(* CODESYS project MC516.project
   CompiledLibraryCompatibilityVersion: LeadSysStudio V3.5 SP15 Patch 4
   Title: MC516

Project tree, tasks and I/O mapping:
  Device : MC516, Leadshine Technology Co., Ltd., order no. 516101, version 3.5.15.40
      settings: RetainMode = 0; RetainStartAddr = 20480; RetainEndAddr = 524288; RetainSize = 524288
    application Application
      libraries: Standard, * (System); VisuDialogs, * (System)
      task EtherCAT_Master_Leadshine_A (cyclic, interval 2000 µs, priority 0) calls EtherCAT_Master_Leadshine_A.EtherCAT_Task, M
      program M [ST]: io, motion, save_check, save_apply, work
      DataMain/
        data type HMIData
        data type SaveData
      function block AxisFB [ST]: calculate_home_delta_μ, follow
      Enum/
        data type State
        data type JogType
      Object/
        data type Button
        data type Cylinder
        data type AxisEC
        data type AxisECFollow
        data type AirBurst
        data type Problem
      function StateNext [ST]
      DataWork/
        data type SupplyData
        data type WorkData
        data type TapData
      function block TapFB [ST]
      visualisation Visualization
      function block SupplyFB [ST]
      Symbols
      function block SimpleMotion [ST]
      trace Trace (task EtherCAT_Master_Leadshine_A): M.tap_data.deviation
      function block AxisFBSetTorqueLimit [ST]
      global variables PersistentVars
    Resource Usage
    Device Diagnose
    Network Configuration
      LocalBus Config
    SoftMotion General Axis Pool
      AxisTap : Axis, 3S - Smart Software Solutions GmbH, order no. 1805, version 4.0.0.0
          settings: wDriveID = 3; eRampType = 3
    High_Speed_IO_Module : High Speed IO, Leadshine Technology Co., Ltd., version 3.5.15.40
        settings: HS_IO_Mode_0.High In IO Mode 0 = 196611; HS_IO_Mode_0.High In IO Mode 2 = 196611; Counter_Mask = 5; Ioin_Mask = 19; HS counter 1.Counter_CountMode = 1; HS counter 2.Counter_CountMode = 1; HS counter 3.Counter_SetWorkMode = 2; HS counter 3.Counter_CountMode = 1; InputFilter Para.Time_In0 = 2; InputFilter Para.Time_In1 = 2; InputFilter Para.Time_In4 = 2
        unmapped channels: Genral_IO_IN, Genral_IO_Out
    LocalBus_Master_Module : LocalBus Master, Leadshine Technology Co., Ltd., version 3.5.15.40
    EtherCAT_Master_Leadshine_A : EtherCAT Master SoftMotion, 3S - Smart Software Solutions GmbH, version 3.5.16.30
        settings: MasterCycleTime = 2000; NetworkName = 'ecat'; SelectNetworkByName = TRUE; SrcAddress1 = 10; SrcAddress2 = 889192738
      XINJE_DS5C1_CoE_Drive_Rev4_0_2 : XINJE-DS5C1 EtherCAT(CoE) Drive Rev4.0 v3.7.70, Xinje Electronics, Inc., order no. XINJE-DS5C1 CoE Drive Rev4.0, version Revision=16#20201207
          settings: Number of Inputs = 6; Number of Infos about Inputs = 6; StationAlias = 4; Sync.Length = 17; FMMU.Length = 17; DC sync0 cycletime = 2000; DC sync1 cycletime = 2000; Number of SDO = 4; Interpolation time period.Value = 2; Homing method.Index = 16#0000; Homing method.Subindex = 16#00; Homing method.Size = 0; Homing method.AbortIfError = FALSE; Homing method.JumpToLine = FALSE; Homing method.Line = 0; Homing method.CompleteAccess = False; RxTxPdo.NumberofEntries = 6; RxTxPdo.Index = 16#1A00; RxTxPdo.DependOnSlot = False; RxTxPdo.DependOnSlotGroup = False; RxTxPdo.OverwrittenByModule = False; Status Word.Offset = 0; Status Word.DependOnSlot = False; Status Word.DependOnSlotGroup = False; ActualPosition.Offset = 0; ActualPosition.DependOnSlot = False; ActualPosition.DependOnSlotGroup = False; Velocity actual value.Offset = 0; Velocity actual value.DependOnSlot = False; Velocity actual value.DependOnSlotGroup = False; ActualTorque.Offset = 0; ActualTorque.DependOnSlot = False; ActualTorque.DependOnSlotGroup = False; ModeOfOperationDisplay.Offset = 0; ModeOfOperationDisplay.DependOnSlot = False; ModeOfOperationDisplay.DependOnSlotGroup = False; Index = 16#5000; SubIndex = 0; Size = 32; Offset = 0;
            DependOnSlot = False; DependOnSlotGroup = False; Status Word.Default = ''; Status Word.Comment = ''; ActualPosition.Default = ''; ActualPosition.Comment = ''; Velocity actual value.Default = ''; Velocity actual value.Comment = ''; ActualTorque.Default = ''; ActualTorque.Comment = ''; ModeOfOperationDisplay.Default = ''; ModeOfOperationDisplay.Comment = ''; Name = 'Encode Single Position'; DataType = 'DINT'; Default = ''; Comment = ''
          unmapped channels: Control Word, TargetPosition, TargetVelocity, TargetTorque, ModeOfOperation, Status Word, ActualPosition, Velocity actual value, ActualTorque, ModeOfOperationDisplay, Encode Single Position
        Axis_2 : Axis, 3S - Smart Software Solutions GmbH, order no. 0, version 4.6.1.0
            settings: wDriveID = 7; dwRatioTechUnitsDenom = 1; eRampType = 3; Number of pulses for one revolution = 131072; The displacement for one revolution of the workbench = 131072; Gear ratio molecule = 1; Gear ratio denominator = 1; ScalingIncs = 131072; AdrOffset_8010 = 36; BitOffset_8010 = 0; BitLength_8010 = 16; Address_8010 = '%QW18'; Type_8010 = 'UINT'; AddressPointer_8010 = ADR(%QW18); AdrOffset_8020 = 40; BitOffset_8020 = 0; BitLength_8020 = 32; Address_8020 = '%QD10'; Type_8020 = 'DINT'; AddressPointer_8020 = ADR(%QD10); AdrOffset_8030 = 44; BitOffset_8030 = 0; BitLength_8030 = 32; Address_8030 = '%QD11'; Type_8030 = 'DINT'; AddressPointer_8030 = ADR(%QD11); AdrOffset_8040 = 48; BitOffset_8040 = 0; BitLength_8040 = 16; Address_8040 = '%QW24'; Type_8040 = 'INT'; AddressPointer_8040 = ADR(%QW24); AdrOffset_8050 = 50; BitOffset_8050 = 0; BitLength_8050 = 8; Address_8050 = '%QB50'; Type_8050 = 'SINT'; AddressPointer_8050 = ADR(%QB50); AdrOffset_8060 = 4294967295; BitOffset_8060 = 0;
              BitLength_8060 = 0; Address_8060 = ''; Type_8060 = ''; AddressPointer_8060 = 0; AdrOffset_8070 = 4294967295; BitOffset_8070 = 0; BitLength_8070 = 0; Address_8070 = ''; Type_8070 = ''; AddressPointer_8070 = 0; AdrOffset_8080 = 4294967295; BitOffset_8080 = 0; BitLength_8080 = 0; Address_8080 = ''; Type_8080 = ''; AddressPointer_8080 = 0; AdrOffset_8090 = 4294967295; BitOffset_8090 = 0; BitLength_8090 = 0; Address_8090 = ''; Type_8090 = ''; AddressPointer_8090 = 0; AdrOffset_8510 = 44; BitOffset_8510 = 0; BitLength_8510 = 16; Address_8510 = '%IW22'; Type_8510 = 'UINT'; AddressPointer_8510 = ADR(%IW22); AdrOffset_8520 = 48; BitOffset_8520 = 0; BitLength_8520 = 32; Address_8520 = '%ID12'; Type_8520 = 'DINT'; AddressPointer_8520 = ADR(%ID12); AdrOffset_8530 = 52; BitOffset_8530 = 0; BitLength_8530 = 32; Address_8530 = '%ID13'; Type_8530 = 'DINT'; AddressPointer_8530 = ADR(%ID13);
              AdrOffset_8540 = 56; BitOffset_8540 = 0; BitLength_8540 = 16; Address_8540 = '%IW28'; Type_8540 = 'INT'; AddressPointer_8540 = ADR(%IW28); AdrOffset_8550 = 58; BitOffset_8550 = 0; BitLength_8550 = 8; Address_8550 = '%IB58'; Type_8550 = 'SINT'; AddressPointer_8550 = ADR(%IB58); AdrOffset_8560 = 4294967295; BitOffset_8560 = 0; BitLength_8560 = 0; Address_8560 = ''; Type_8560 = ''; AddressPointer_8560 = 0; AdrOffset_8570 = 4294967295; BitOffset_8570 = 0; BitLength_8570 = 0; Address_8570 = ''; Type_8570 = ''; AddressPointer_8570 = 0; AdrOffset_8580 = 4294967295; BitOffset_8580 = 0; BitLength_8580 = 0; Address_8580 = ''; Type_8580 = ''; AddressPointer_8580 = 0; AdrOffset_8590 = 4294967295; BitOffset_8590 = 0; BitLength_8590 = 0; Address_8590 = ''; Type_8590 = ''; AddressPointer_8590 = 0; AdrOffset_8600 = 4294967295; BitOffset_8600 = 0; BitLength_8600 = 0; Address_8600 = '';
              Type_8600 = ''; AddressPointer_8600 = 0; AdrOffset_8600 = 4294967295; BitOffset_8600 = 0; BitLength_8600 = 0; Address_8610 = ''; Type_8610 = ''; AddressPointer_8610 = 0; AdrOffset_8620 = 4294967295; BitOffset_8620 = 0; BitLength_8620 = 0; Address_8620 = ''; Type_8620 = ''; AddressPointer_8620 = 0
      XINJE_DS5C1_CoE_Drive_Rev4_0_1 : XINJE-DS5C1 EtherCAT(CoE) Drive Rev4.0 v3.7.70, Xinje Electronics, Inc., order no. XINJE-DS5C1 CoE Drive Rev4.0, version Revision=16#20201207
          settings: Number of Inputs = 6; Number of Infos about Inputs = 6; StationAlias = 3; Sync.Length = 17; FMMU.Length = 17; DC sync0 cycletime = 2000; DC sync1 cycletime = 2000; Number of SDO = 4; Interpolation time period.Value = 2; Homing method.Index = 16#0000; Homing method.Subindex = 16#00; Homing method.Size = 0; Homing method.AbortIfError = FALSE; Homing method.JumpToLine = FALSE; Homing method.Line = 0; Homing method.CompleteAccess = False; RxTxPdo.NumberofEntries = 6; RxTxPdo.Index = 16#1A00; RxTxPdo.DependOnSlot = False; RxTxPdo.DependOnSlotGroup = False; RxTxPdo.OverwrittenByModule = False; Status Word.Offset = 0; Status Word.DependOnSlot = False; Status Word.DependOnSlotGroup = False; ActualPosition.Offset = 0; ActualPosition.DependOnSlot = False; ActualPosition.DependOnSlotGroup = False; Velocity actual value.Offset = 0; Velocity actual value.DependOnSlot = False; Velocity actual value.DependOnSlotGroup = False; ActualTorque.Offset = 0; ActualTorque.DependOnSlot = False; ActualTorque.DependOnSlotGroup = False; ModeOfOperationDisplay.Offset = 0; ModeOfOperationDisplay.DependOnSlot = False; ModeOfOperationDisplay.DependOnSlotGroup = False; Index = 16#5000; SubIndex = 0; Size = 32; Offset = 0;
            DependOnSlot = False; DependOnSlotGroup = False; Status Word.Default = ''; Status Word.Comment = ''; ActualPosition.Default = ''; ActualPosition.Comment = ''; Velocity actual value.Default = ''; Velocity actual value.Comment = ''; ActualTorque.Default = ''; ActualTorque.Comment = ''; ModeOfOperationDisplay.Default = ''; ModeOfOperationDisplay.Comment = ''; Name = 'Encode Single Position'; DataType = 'DINT'; Default = ''; Comment = ''
          unmapped channels: Control Word, TargetPosition, TargetVelocity, TargetTorque, ModeOfOperation, Status Word, ActualPosition, Velocity actual value, ActualTorque, ModeOfOperationDisplay, Encode Single Position
        Axis_1 : Axis, 3S - Smart Software Solutions GmbH, order no. 0, version 4.6.1.0
            settings: wDriveID = 6; dwRatioTechUnitsDenom = 1; eRampType = 3; Number of pulses for one revolution = 131072; The displacement for one revolution of the workbench = 131072; Gear ratio molecule = 1; Gear ratio denominator = 1; ScalingIncs = 131072; AdrOffset_8010 = 20; BitOffset_8010 = 0; BitLength_8010 = 16; Address_8010 = '%QW10'; Type_8010 = 'UINT'; AddressPointer_8010 = ADR(%QW10); AdrOffset_8020 = 24; BitOffset_8020 = 0; BitLength_8020 = 32; Address_8020 = '%QD6'; Type_8020 = 'DINT'; AddressPointer_8020 = ADR(%QD6); AdrOffset_8030 = 28; BitOffset_8030 = 0; BitLength_8030 = 32; Address_8030 = '%QD7'; Type_8030 = 'DINT'; AddressPointer_8030 = ADR(%QD7); AdrOffset_8040 = 32; BitOffset_8040 = 0; BitLength_8040 = 16; Address_8040 = '%QW16'; Type_8040 = 'INT'; AddressPointer_8040 = ADR(%QW16); AdrOffset_8050 = 34; BitOffset_8050 = 0; BitLength_8050 = 8; Address_8050 = '%QB34'; Type_8050 = 'SINT'; AddressPointer_8050 = ADR(%QB34); AdrOffset_8060 = 4294967295; BitOffset_8060 = 0;
              BitLength_8060 = 0; Address_8060 = ''; Type_8060 = ''; AddressPointer_8060 = 0; AdrOffset_8070 = 4294967295; BitOffset_8070 = 0; BitLength_8070 = 0; Address_8070 = ''; Type_8070 = ''; AddressPointer_8070 = 0; AdrOffset_8080 = 4294967295; BitOffset_8080 = 0; BitLength_8080 = 0; Address_8080 = ''; Type_8080 = ''; AddressPointer_8080 = 0; AdrOffset_8090 = 4294967295; BitOffset_8090 = 0; BitLength_8090 = 0; Address_8090 = ''; Type_8090 = ''; AddressPointer_8090 = 0; AdrOffset_8510 = 24; BitOffset_8510 = 0; BitLength_8510 = 16; Address_8510 = '%IW12'; Type_8510 = 'UINT'; AddressPointer_8510 = ADR(%IW12); AdrOffset_8520 = 28; BitOffset_8520 = 0; BitLength_8520 = 32; Address_8520 = '%ID7'; Type_8520 = 'DINT'; AddressPointer_8520 = ADR(%ID7); AdrOffset_8530 = 32; BitOffset_8530 = 0; BitLength_8530 = 32; Address_8530 = '%ID8'; Type_8530 = 'DINT'; AddressPointer_8530 = ADR(%ID8);
              AdrOffset_8540 = 36; BitOffset_8540 = 0; BitLength_8540 = 16; Address_8540 = '%IW18'; Type_8540 = 'INT'; AddressPointer_8540 = ADR(%IW18); AdrOffset_8550 = 38; BitOffset_8550 = 0; BitLength_8550 = 8; Address_8550 = '%IB38'; Type_8550 = 'SINT'; AddressPointer_8550 = ADR(%IB38); AdrOffset_8560 = 4294967295; BitOffset_8560 = 0; BitLength_8560 = 0; Address_8560 = ''; Type_8560 = ''; AddressPointer_8560 = 0; AdrOffset_8570 = 4294967295; BitOffset_8570 = 0; BitLength_8570 = 0; Address_8570 = ''; Type_8570 = ''; AddressPointer_8570 = 0; AdrOffset_8580 = 4294967295; BitOffset_8580 = 0; BitLength_8580 = 0; Address_8580 = ''; Type_8580 = ''; AddressPointer_8580 = 0; AdrOffset_8590 = 4294967295; BitOffset_8590 = 0; BitLength_8590 = 0; Address_8590 = ''; Type_8590 = ''; AddressPointer_8590 = 0; AdrOffset_8600 = 4294967295; BitOffset_8600 = 0; BitLength_8600 = 0; Address_8600 = '';
              Type_8600 = ''; AddressPointer_8600 = 0; AdrOffset_8600 = 4294967295; BitOffset_8600 = 0; BitLength_8600 = 0; Address_8610 = ''; Type_8610 = ''; AddressPointer_8610 = 0; AdrOffset_8620 = 4294967295; BitOffset_8620 = 0; BitLength_8620 = 0; Address_8620 = ''; Type_8620 = ''; AddressPointer_8620 = 0
      XINJE_DS5C1_CoE_Drive_Rev4_0 : XINJE-DS5C1 EtherCAT(CoE) Drive Rev4.0 v3.7.70, Xinje Electronics, Inc., order no. XINJE-DS5C1 CoE Drive Rev4.0, version Revision=16#20201207
          settings: Number of Inputs = 6; Number of Infos about Inputs = 6; StationAlias = 1; Sync.Length = 17; FMMU.Length = 17; DC sync0 cycletime = 2000; DC sync1 cycletime = 2000; Number of SDO = 4; Interpolation time period.Value = 2; Homing method.Index = 16#0000; Homing method.Subindex = 16#00; Homing method.Size = 0; Homing method.AbortIfError = FALSE; Homing method.JumpToLine = FALSE; Homing method.Line = 0; Homing method.CompleteAccess = False; RxTxPdo.NumberofEntries = 6; RxTxPdo.Index = 16#1A00; RxTxPdo.DependOnSlot = False; RxTxPdo.DependOnSlotGroup = False; RxTxPdo.OverwrittenByModule = False; Status Word.Offset = 0; Status Word.DependOnSlot = False; Status Word.DependOnSlotGroup = False; ActualPosition.Offset = 0; ActualPosition.DependOnSlot = False; ActualPosition.DependOnSlotGroup = False; Velocity actual value.Offset = 0; Velocity actual value.DependOnSlot = False; Velocity actual value.DependOnSlotGroup = False; ActualTorque.Offset = 0; ActualTorque.DependOnSlot = False; ActualTorque.DependOnSlotGroup = False; ModeOfOperationDisplay.Offset = 0; ModeOfOperationDisplay.DependOnSlot = False; ModeOfOperationDisplay.DependOnSlotGroup = False; Index = 16#5000; SubIndex = 0; Size = 32; Offset = 0;
            DependOnSlot = False; DependOnSlotGroup = False; Status Word.Default = ''; Status Word.Comment = ''; ActualPosition.Default = ''; ActualPosition.Comment = ''; Velocity actual value.Default = ''; Velocity actual value.Comment = ''; ActualTorque.Default = ''; ActualTorque.Comment = ''; ModeOfOperationDisplay.Default = ''; ModeOfOperationDisplay.Comment = ''; Name = 'Encode Single Position'; DataType = 'DINT'; Default = ''; Comment = ''
          unmapped channels: Control Word, TargetPosition, TargetVelocity, TargetTorque, ModeOfOperation, Status Word, ActualPosition, Velocity actual value, ActualTorque, ModeOfOperationDisplay, Encode Single Position
        Axis : Axis, 3S - Smart Software Solutions GmbH, order no. 0, version 4.6.1.0
            settings: wDriveID = 4; dwRatioTechUnitsDenom = 1; eRampType = 3; Number of pulses for one revolution = 131072; The displacement for one revolution of the workbench = 131072; Gear ratio molecule = 1; Gear ratio denominator = 1; ScalingIncs = 131072; AdrOffset_8010 = 4; BitOffset_8010 = 0; BitLength_8010 = 16; Address_8010 = '%QW2'; Type_8010 = 'UINT'; AddressPointer_8010 = ADR(%QW2); AdrOffset_8020 = 8; BitOffset_8020 = 0; BitLength_8020 = 32; Address_8020 = '%QD2'; Type_8020 = 'DINT'; AddressPointer_8020 = ADR(%QD2); AdrOffset_8030 = 12; BitOffset_8030 = 0; BitLength_8030 = 32; Address_8030 = '%QD3'; Type_8030 = 'DINT'; AddressPointer_8030 = ADR(%QD3); AdrOffset_8040 = 16; BitOffset_8040 = 0; BitLength_8040 = 16; Address_8040 = '%QW8'; Type_8040 = 'INT'; AddressPointer_8040 = ADR(%QW8); AdrOffset_8050 = 18; BitOffset_8050 = 0; BitLength_8050 = 8; Address_8050 = '%QB18'; Type_8050 = 'SINT'; AddressPointer_8050 = ADR(%QB18); AdrOffset_8060 = 4294967295; BitOffset_8060 = 0;
              BitLength_8060 = 0; Address_8060 = ''; Type_8060 = ''; AddressPointer_8060 = 0; AdrOffset_8070 = 4294967295; BitOffset_8070 = 0; BitLength_8070 = 0; Address_8070 = ''; Type_8070 = ''; AddressPointer_8070 = 0; AdrOffset_8080 = 4294967295; BitOffset_8080 = 0; BitLength_8080 = 0; Address_8080 = ''; Type_8080 = ''; AddressPointer_8080 = 0; AdrOffset_8090 = 4294967295; BitOffset_8090 = 0; BitLength_8090 = 0; Address_8090 = ''; Type_8090 = ''; AddressPointer_8090 = 0; AdrOffset_8510 = 4; BitOffset_8510 = 0; BitLength_8510 = 16; Address_8510 = '%IW2'; Type_8510 = 'UINT'; AddressPointer_8510 = ADR(%IW2); AdrOffset_8520 = 8; BitOffset_8520 = 0; BitLength_8520 = 32; Address_8520 = '%ID2'; Type_8520 = 'DINT'; AddressPointer_8520 = ADR(%ID2); AdrOffset_8530 = 12; BitOffset_8530 = 0; BitLength_8530 = 32; Address_8530 = '%ID3'; Type_8530 = 'DINT'; AddressPointer_8530 = ADR(%ID3);
              AdrOffset_8540 = 16; BitOffset_8540 = 0; BitLength_8540 = 16; Address_8540 = '%IW8'; Type_8540 = 'INT'; AddressPointer_8540 = ADR(%IW8); AdrOffset_8550 = 18; BitOffset_8550 = 0; BitLength_8550 = 8; Address_8550 = '%IB18'; Type_8550 = 'SINT'; AddressPointer_8550 = ADR(%IB18); AdrOffset_8560 = 4294967295; BitOffset_8560 = 0; BitLength_8560 = 0; Address_8560 = ''; Type_8560 = ''; AddressPointer_8560 = 0; AdrOffset_8570 = 4294967295; BitOffset_8570 = 0; BitLength_8570 = 0; Address_8570 = ''; Type_8570 = ''; AddressPointer_8570 = 0; AdrOffset_8580 = 4294967295; BitOffset_8580 = 0; BitLength_8580 = 0; Address_8580 = ''; Type_8580 = ''; AddressPointer_8580 = 0; AdrOffset_8590 = 4294967295; BitOffset_8590 = 0; BitLength_8590 = 0; Address_8590 = ''; Type_8590 = ''; AddressPointer_8590 = 0; AdrOffset_8600 = 4294967295; BitOffset_8600 = 0; BitLength_8600 = 0; Address_8600 = '';
              Type_8600 = ''; AddressPointer_8600 = 0; AdrOffset_8600 = 4294967295; BitOffset_8600 = 0; BitLength_8600 = 0; Address_8610 = ''; Type_8610 = ''; AddressPointer_8610 = 0; AdrOffset_8620 = 4294967295; BitOffset_8620 = 0; BitLength_8620 = 0; Address_8620 = ''; Type_8620 = ''; AddressPointer_8620 = 0
  text list GlobalTextList
*)

// Device/Application/DataMain/HMIData
{ attribute 'pack_mode' := ''}
TYPE HMIData :
STRUCT
	//
	sv: SaveData;
	sv_trigger: BOOL;
	sv_need_check: BOOL;
	sv_need: BOOL;
	//
	plc_ready: BOOL;
	hmi_ready: BOOL;
	run: BOOL;
	stop: BOOL;
	home: BOOL;
	problem_fix: ARRAY[0..7] OF BOOL;
	//
	supply_test: BOOL;
	supply_clamp: BOOL;
	supply_extract_down: BOOL;
	supply_extract_pull: BOOL;
	tap_lubricate: BOOL;
	supply_clean: BOOL;
	jog_micro_per_sec_or_rev: UINT;
	jog_n: BOOL;
	jog_p: BOOL;
	//
	view_input: ARRAY[0..15] OF BOOL;
	view_output: ARRAY[0..15] OF BOOL;
	//
	view_can_run: BOOL;
	view_can_stop: BOOL;
	view_can_home: BOOL;
	view_auto: BOOL;
	view_manual: BOOL;
	//
	view_axis_encoder: ARRAY[0..2] OF DINT;
	view_axis_micro: ARRAY[0..2] OF DINT;
	view_axis_mNm: ARRAY[0..2] OF UDINT;
	//
	view_load: UINT;
	view_problem: ARRAY[0..7] OF BOOL;
	view_tap_deviation_micron: UINT;
	view_cycle_count: UDINT;
	view_cycle_time_msec: UDINT;
	//
	view_state: ARRAY[0..4] OF INT;
END_STRUCT
END_TYPE

// Device/Application/DataMain/SaveData
{ attribute 'pack_mode' := ''}
TYPE SaveData :
STRUCT
	set_done: BOOL;
	////////
	//SAME//
	////////
	cylinder_n_delay_msec: ARRAY[0..2] OF UINT;
	cylinder_p_delay_msec: ARRAY[0..2] OF UINT;
	air_burst_delay_msec: ARRAY[0..1] OF UINT;
	//
	// (a) increments        <> (d) motor turns
	// (b) motor turns       <> (e) gear output turns
	// (c) gear output turns <> (f) units in application
	// .iRatioTechUnitsNum = gear_num = gear_dir * d * e * f 
	// .dwRatioTechUnitsDenom = gear_den = a * b * c
	max_rpm: ARRAY[0..2] OF UINT;
	gear_num: ARRAY[0..2] OF DINT;
	gear_den: ARRAY[0..2] OF DINT;
	gear_dir: ARRAY[0..2] OF BOOL;
	home_torque_mNm: ARRAY[0..2] OF UINT;
	home_encoder_value_recorded: BOOL;
	home_encoder_value: ARRAY[0..2] OF DINT;
	max_micro_recorded: BOOL;
	max_micro: ARRAY[0..2] OF DINT;
	overload_hold_torque_factor: ARRAY[0..2] OF UINT;
	overload_hold_torque_time_msec: ARRAY[0..2] OF UINT;
	overload_instant_torque_factor: ARRAY[0..2] OF UINT;
	ramp_time_msec: ARRAY[0..2] OF UINT;
	jerk_factor: ARRAY[0..2] OF UINT;
	///////////
	//MACHINE//
	///////////
	supply_micro_per_sec: UDINT;
	//
	tap_begin_micron: UDINT; // vị trí bắt đầu taro
	tap_depth_micron: UDINT; // độ sâu từ vị trí bắt đầu taro
	tap_micron_per_rev: UDINT; // bước ren μm
	tap_rpm: UDINT; // tốc độ taro
	tap_backlash_micro: UINT; // độ rơ micro vòng
	tap_deviation_micron_max: UINT;
END_STRUCT
END_TYPE

// Device/Application/Enum/State
{attribute 'qualified_only'}
{attribute 'strict'}
TYPE State :
(
	NONE := 0,
	RST := 1,
	RST_DONE := 50,
	HOME := 51,
	HOME_FORWARD := 71,
	HOME_DONE := 90,
	HOME_OFFSET := 91,
	HOME_OFFSET_DONE := 99,
	READY := 100,
	RUN := 101,
	RUN_ING := 200
);
END_TYPE

// Device/Application/Object/Button
{ attribute 'pack_mode' := ''}
TYPE Button :
STRUCT
	on: BOOL;
	rise: R_TRIG;
	rise_physical: R_TRIG;
	fall: F_TRIG;
	fall_physical: F_TRIG;
	timer: TON;
END_STRUCT
END_TYPE

// Device/Application/Object/Cylinder
{ attribute 'pack_mode' := ''}
TYPE Cylinder :
STRUCT
	on: BOOL;
	n_timer: TON;
	p_timer: TON;
END_STRUCT
END_TYPE

// Device/Application/Object/AxisEC
{ attribute 'pack_mode' := ''}
TYPE AxisEC :
STRUCT
	///////
	//REF//
	///////
	ref: POINTER TO SM3_Drive_ETC_DS402_CyclicSync.AXIS_REF_ETC_DS402_CS;
	read: POINTER TO SMC3_ETC_ReadParameter_CoE;
	write: POINTER TO SMC3_ETC_WriteParameter_CoE;
	read_status: POINTER TO MC_ReadStatus;
	set_mode: POINTER TO SMC_SetControllerMode;
	power: POINTER TO MC_Power;
	reset: POINTER TO MC_Reset;
	stop: POINTER TO MC_Stop;
	inch: POINTER TO SMC_Inch;
	fsv: POINTER TO SMC_FollowSetValues;
	sp: POINTER TO MC_SetPosition;
	mabs: POINTER TO MC_MoveAbsolute;
	set_torque_limit: AxisFBSetTorqueLimit;
	////////
	//DATA//
	////////
	encoder_resolution: DINT;
	torque_rated_Nm: LREAL;
	encoder_single_position: DINT;
	///////////
	//PROCESS//
	///////////
	state: INT;
	torque_Nm: LREAL;
	torque_Nm_abs: LREAL;
	overload: BOOL;
	overload_check: BOOL;
	overload_hold_torque_Nm: LREAL;
	overload_hold_torque_timer: TON;
	overload_instant_torque_Nm: LREAL;
	//home
	home_done: BOOL; // = TRUE khi về gốc thành công, chỉ về gốc khi bật máy
	home_done_forward_ignore: BOOL;
	home_to_encoder: BOOL; //
	home_torque_Nm: LREAL;
	home_hit_timer: TON;
	home_hit_test: BOOL;
	home_offset_absolute_μ: LREAL; // vị trí từ điểm va chạm đến gốc tuyệt đối, xem hàm save_apply()
	home_back_μ_per_sec: LREAL; // tốc độ lùi về lấy gốc
	home_forward_μ_per_sec: LREAL; // tốc độ tiến sau khi lấy gốc xong
	home_offset_μ: LREAL; // giá trị này để thực hiện lệnh state = State.HOME_OFFSET ở trong AxisLinearFB
	home_encoder_value_recorded: BOOL;
	home_encoder_value_save: POINTER TO DINT; // pointer tới giá trị ở save data
	home_encoder_delta: DINT;
	home_delta_μ: LREAL;
	//
	ramp_time_sec: LREAL;
	jerk_factor: LREAL;
	//
	jog_type: JogType;
	jog_delta: LREAL;
	jog_velocity: LREAL;
	jog_acceleration: LREAL;
	max_μ_recorded: BOOL;
	max_μ_save: POINTER TO DINT;
	max_μ: LREAL; // giới hạn vị trí tối đa có thể di chuyển từ gốc tuyệt đối
	max_μ_per_sec: LREAL; // giới hạn tốc độ tối đa
	//run
	target_position_μ: LREAL; // sử dụng cho state = State.RUN ở trong AxisLinearFB
	target_velocity_μ_per_sec: LREAL; // sử dụng cho state = State.RUN ở trong AxisLinearFB
END_STRUCT
END_TYPE

// Device/Application/DataWork/SupplyData
{ attribute 'pack_mode' := ''}
TYPE SupplyData :
STRUCT
	state: INT;
	state_extract: INT;
	axis: AxisEC;
	axis_fb: AxisFB;
	//
	input_air: BOOL;
	input_foil: BOOL;
	//
	no_air: Problem;
	foil_stuck: Problem;
	clamp: Cylinder;
	extract_down: Cylinder;
	extract_pull: Cylinder;
	clean: AirBurst;
	//
	index_count: LREAL;
	μ_per_sec: LREAL;
END_STRUCT
END_TYPE

// Device/Application/DataWork/WorkData
{ attribute 'pack_mode' := ''}
TYPE WorkData :
STRUCT
	state: INT;
	//
	input_run: Button;
	input_stop: Button;
	input_home: Button;
	//
	can_run: BOOL;
	can_stop: BOOL;
	can_home: BOOL;
	auto: Button;
	overload: Problem;
	alarm: BOOL;
	//
	supply_test: Button;
	//
	manual: BOOL;
	cycle_start_msec: ULINT;
	cycle_time_msec: UDINT;
END_STRUCT
END_TYPE

// Device/Application/DataWork/TapData
{ attribute 'pack_mode' := ''}
TYPE TapData :
STRUCT
	state: INT;
	axis_move: AxisEC;
	axis_move_fb: AxisFB;
	axis_move_follow_data: AxisECFollow;
	axis_spin: AxisEC;
	axis_spin_fb: AxisFB;
	axis_spin_follow_data: AxisECFollow;
	//
	axis_v: POINTER TO SM3_Basic.AXIS_REF_VIRTUAL_SM3;
	axis_v_power: MC_Power;
	axis_v_stop: MC_Stop;
	axis_v_inch: SMC_Inch;
	axis_v_sp: MC_SetPosition;
	axis_v_mabs: MC_MoveAbsolute;
	//
	begin_μm: LREAL;
	depth_μm: LREAL;
	μm_per_rev: LREAL;
	rps: LREAL;
	backlash_μ: LREAL;
	//
	lubricate: AirBurst;
	//
	deviation_μm: LREAL;
	deviation_μm_max: LREAL;
	deviation_overload: BOOL;
	//
	load: LREAL;
	load_sum: LREAL;
	load_count: LREAL;
	time_delta_sec: LREAL;
END_STRUCT
END_TYPE

// Device/Application/Object/AxisECFollow
TYPE AxisECFollow :
STRUCT
	target: POINTER TO SM3_Basic.AXIS_REF_SM3;
	ratio: LREAL;
	offset: LREAL;
	offset_motion: SimpleMotion;
	//
	self_begin: LREAL;
	target_begin: LREAL;
	target_delta: LREAL;
	//
	deviation: LREAL;
END_STRUCT
END_TYPE

// Device/Application/Object/AirBurst
TYPE AirBurst :
STRUCT
	on: BOOL;
	timer: TON;
END_STRUCT
END_TYPE

// Device/Application/Enum/JogType
{attribute 'qualified_only'}
{attribute 'strict'}
TYPE JogType :
(
	NONE := 0,
	INCH := 1, // inch function
	FSV := 2 // follow set value function
);
END_TYPE

// Device/Application/Object/Problem
TYPE Problem :
STRUCT
	on: BOOL;
	timer: TON;
	rise: R_TRIG;
	fix_rise: R_TRIG;
END_STRUCT
END_TYPE

// Device/Application/PersistentVars
{attribute 'qualified_only'}
VAR_GLOBAL PERSISTENT RETAIN
END_VAR
VAR_GLOBAL PERSISTENT
	M.save: SaveData;
END_VAR

// Device/Application/M
PROGRAM M
VAR
	time_msec_last: ULINT;
	time_msec : ULINT;
	time_delta_sec: LREAL;
	//
	axiss: ARRAY [0..2] OF POINTER TO SM3_Drive_ETC_DS402_CyclicSync.AXIS_REF_ETC_DS402_CS;
	// dùng pointer để dễ dàng thao tác với nhiều trục hơn, xem hàm motion()
	axiss_read: ARRAY[0..2] OF SMC3_ETC_ReadParameter_CoE;
	axiss_write: ARRAY[0..2] OF SMC3_ETC_WriteParameter_CoE;
	axiss_read_status: ARRAY[0..2] OF MC_ReadStatus;
	axiss_change_gearing_ratio: ARRAY[0..2] OF SMC_ChangeGearingRatio;
	axiss_reinit_drive: ARRAY[0..2] OF SMC3_ReinitDrive;
	axiss_set_mode: ARRAY[0..2] OF SMC_SetControllerMode;
	axiss_power: ARRAY[0..2] OF MC_Power; // bật tắt động cơ
	axiss_reset: ARRAY[0..2] OF MC_Reset; // reset lỗi
	axiss_stop: ARRAY[0..2] OF MC_Stop; // dừng
	axiss_inch: ARRAY[0..2] OF SMC_Inch;
	axiss_fsv: ARRAY[0..2] OF SMC_FollowSetValues;
	axiss_sp: ARRAY[0..2] OF MC_SetPosition;
	axiss_mabs: ARRAY[0..2] OF MC_MoveAbsolute;
	axiss_encoder_resolution: ARRAY[0..2] OF DINT;
	axiss_rated_torque_Nm: ARRAY[0..2] OF LREAL;
	axiss_max_rpm: ARRAY[0..2] OF UINT;
	axiss_max_μ_per_sec: ARRAY[0..2] OF LREAL;
	axiss_ready_all: BOOL;
	//
	state_main: INT;
	motion_active: BOOL;
	main_save: Button;
	supply_data: SupplyData;
	supply_fb: SupplyFB;
	tap_data: TapData;
	tap_fb: TapFB;
	work_data: WorkData;
	hmi: HMIData;
	//
	i: INT;
	j: INT;
	k: INT;
	axis_ec_i: POINTER TO AxisEC;
	axis_fb_i: POINTER TO AxisFB;
	cylinder_i: POINTER TO Cylinder;
	air_burst_i: POINTER TO AirBurst;
	//
	test: BOOL;
END_VAR

VAR CONSTANT
	c_axis_i_max: INT := 3 - 1;
	c_cylinder_i_max: INT := 3 - 1;
	c_air_burst_i_max: INT := 2 - 1;
END_VAR

VAR RETAIN
	cycle_count: UDINT;
	cycle_count_reset_time_msec: ULINT;
END_VAR

VAR PERSISTENT
	save: SaveData;
END_VAR

MC_SysLib.SysTimeRtc.SysTimeRtcHighResGet(pTimestamp:= time_msec);
time_delta_sec := ULINT_TO_LREAL(time_msec - time_msec_last) * 1E-3;
time_msec_last := time_msec;
hmi.view_state[0] := state_main;
IF motion_active THEN
	motion();
END_IF
CASE state_main OF
	State.NONE: // khi khởi động thì state_main = 0 tức là = State.NONE
		axiss[0] := ADR(Axis); // k = ADR(x) viết tắt cho "address of x" là hàm để lấy giá trị con trỏ (pointer) về biến x
		axiss[1] := ADR(Axis_1); // ví dụ muốn thay đổi giá trị của x ta sẽ viết k^ = 12345
		axiss[2] := ADR(Axis_2);
		axiss_change_gearing_ratio[0].iMovementType := SMC_MOVEMENTTYPE.rotary;
		axiss_change_gearing_ratio[1].iMovementType := SMC_MOVEMENTTYPE.linear;
		axiss_change_gearing_ratio[2].iMovementType := SMC_MOVEMENTTYPE.linear;
		axiss_change_gearing_ratio[0].fPositionPeriod := 1_000;
		axiss_change_gearing_ratio[1].fPositionPeriod := 1_000;
		axiss_change_gearing_ratio[2].fPositionPeriod := 1_000;
		tap_data.axis_v := ADR(AxisTap);
		motion_active := FALSE;
		test := FALSE;
		StateNext(state_main); // chuyển tới trạng thái tiếp theo
	1:
		FOR i := 0 TO c_axis_i_max BY 1 DO // hàm FOR, FOR i = 0 TO 3 BY 1 DO sẽ chạy 4 lần i = [0, 1, 2, 3]
			CASE i OF // hàm CASE, lựa chọn theo giá trị i
				0:
					axis_ec_i := ADR(supply_data.axis);
					axis_fb_i := ADR(supply_data.axis_fb);
				1:
					axis_ec_i := ADR(tap_data.axis_move);
					axis_fb_i := ADR(tap_data.axis_move_fb);
				2:
					axis_ec_i := ADR(tap_data.axis_spin);
					axis_fb_i := ADR(tap_data.axis_spin_fb);
			END_CASE
			axis_ec_i^.ref := axiss[i];
			axis_ec_i^.read := ADR(axiss_read[i]);
			axis_ec_i^.write := ADR(axiss_write[i]);
			axis_ec_i^.read_status := ADR(axiss_read_status[i]);
			axis_ec_i^.set_mode := ADR(axiss_set_mode[i]);
			axis_ec_i^.power := ADR(axiss_power[i]);
			axis_ec_i^.reset := ADR(axiss_reset[i]);
			axis_ec_i^.stop := ADR(axiss_stop[i]);
			axis_ec_i^.inch := ADR(axiss_inch[i]);
			axis_ec_i^.fsv := ADR(axiss_fsv[i]);
			axis_ec_i^.sp := ADR(axiss_sp[i]);
			axis_ec_i^.mabs := ADR(axiss_mabs[i]);
			axis_fb_i^.d := axis_ec_i;
		END_FOR
		StateNext(state_main);
	2:
		axiss_ready_all := TRUE; // biến tạm thời để kiểm tra tất cả các servo đã hoàn thành lệnh hay chưa
		FOR i := 0 TO c_axis_i_max BY 1 DO
			axiss_ready_all := axiss_ready_all AND axiss[i]^.wCommunicationState = 100;
		END_FOR
		IF axiss_ready_all THEN // hoàn thành kết nối tất cả servo, ta đên bước tiếp theo
			motion_active := TRUE;
			state_main := 11;
		END_IF
	11: // đọc số xung encoder của servo
		FOR i := 0 TO c_axis_i_max BY 1 DO
			axiss_read[i].uiIndex := 16#608F; // mở ETHERCAT/XINJE_DS5C1.../ xem trong mục "CoE Online"
			axiss_read[i].usiSubIndex := 1; //
			axiss_read[i].xExecute := TRUE;
		END_FOR
		StateNext(state_main);
	12:
		axiss_ready_all := TRUE;
		FOR i := 0 TO c_axis_i_max BY 1 DO
			axiss_ready_all := axiss_ready_all AND axiss_read[i].xDone;
		END_FOR
		IF axiss_ready_all THEN
			FOR i := 0 TO c_axis_i_max BY 1 DO
				axiss_read[i].xExecute := FALSE;
				// Sau thực hiện hàm thành công phải đặt Execute = FALSE để cho lần đọc tiếp theo
				// vì đa số hàm chỉ chạy khi Execute chuyển từ FALSE sang TRUE (Rising edge)
				// xem Defination của hàm đê biết thêm chi tiết
				axiss_encoder_resolution[i] := DWORD_TO_DINT(axiss_read[i].dwValue);
			END_FOR
			StateNext(state_main);
		END_IF
	13: // đọc momen max của servo
		FOR i := 0 TO c_axis_i_max BY 1 DO
			axiss_read[i].uiIndex := 16#6076;
			axiss_read[i].usiSubIndex := 0;
			axiss_read[i].xExecute := TRUE;
		END_FOR
		StateNext(state_main);
	14:
		axiss_ready_all := TRUE;
		FOR i := 0 TO c_axis_i_max BY 1 DO
			axiss_ready_all := axiss_ready_all AND axiss_read[i].xDone;
		END_FOR
		IF axiss_ready_all THEN
			FOR i := 0 TO c_axis_i_max BY 1 DO
				axiss_read[i].xExecute := FALSE;
				axiss_rated_torque_Nm[i] := DWORD_TO_LREAL(axiss_read[i].dwValue) * 1E-3;
			END_FOR
			StateNext(state_main);
		END_IF
	15: // đọc max rpm của servo
		FOR i := 0 TO c_axis_i_max BY 1 DO
			axiss_read[i].uiIndex := 16#6080;
			axiss_read[i].usiSubIndex := 0;
			axiss_read[i].xExecute := TRUE;
		END_FOR
		StateNext(state_main);
	16:
		axiss_ready_all := TRUE;
		FOR i := 0 TO c_axis_i_max BY 1 DO
			axiss_ready_all := axiss_ready_all AND axiss_read[i].xDone;
		END_FOR
		IF axiss_ready_all THEN
			FOR i := 0 TO c_axis_i_max BY 1 DO
				axiss_read[i].xExecute := FALSE;
				axiss_max_rpm[i] := DWORD_TO_UINT(axiss_read[i].dwValue);
			END_FOR
			StateNext(state_main);
		END_IF
	17:
		FOR i := 0 TO c_axis_i_max BY 1 DO
			CASE i OF
				0: axis_ec_i := ADR(supply_data.axis);
				1: axis_ec_i := ADR(tap_data.axis_move);
				2: axis_ec_i := ADR(tap_data.axis_spin);
			END_CASE
			axis_ec_i^.encoder_resolution := axiss_encoder_resolution[i];
			axis_ec_i^.torque_rated_Nm := axiss_rated_torque_Nm[i];
		END_FOR
		IF NOT save.set_done THEN
			save.set_done := TRUE;
			//
			FOR i := 0 TO c_cylinder_i_max DO
				save.cylinder_n_delay_msec[i] := 0_200 + INT_TO_UINT(i * 2);
				save.cylinder_p_delay_msec[i] := 0_200 + INT_TO_UINT(i * 2 + 1);
			END_FOR
			FOR i := 0 TO c_air_burst_i_max DO
				save.air_burst_delay_msec[i] := 0_200 + INT_TO_UINT(i);
			END_FOR
			//
			save.home_encoder_value_recorded := FALSE;
			save.max_micro_recorded := TRUE;
			FOR i := 0 TO c_axis_i_max BY 1 DO
				save.max_rpm[i] := 3000;
				save.gear_dir[i] := TRUE;
				save.gear_num[i] := axiss_encoder_resolution[i] / 2;
				save.gear_den[i] := axiss_encoder_resolution[i];
				save.home_torque_mNm[i] := 0_797; // 100 kg of force with 5mm ball screw
				save.home_encoder_value[i] := 0;
				save.max_micro[i] := 80_000;
				save.overload_hold_torque_factor[i] := 0_900 + INT_TO_UINT(i);
				save.overload_hold_torque_time_msec[i] := 1_000 + INT_TO_UINT(i);
				save.overload_instant_torque_factor[i] := 2_900 + INT_TO_UINT(i);
				save.ramp_time_msec[i] := 0_100;
				save.jerk_factor[i] := 30;
			END_FOR
			//
			save.supply_micro_per_sec := 1_000;
		END_IF
		StateNext(state_main);
	18:// set gear
		FOR i := 0 TO c_axis_i_max BY 1 DO
			axiss_change_gearing_ratio[i].iRatioTechUnitsNum := (BOOL_TO_DINT(save.gear_dir[i]) * 2 - 1) * save.gear_num[i];
			axiss_change_gearing_ratio[i].dwRatioTechUnitsDenom := DINT_TO_DWORD(save.gear_den[i]);
			axiss_change_gearing_ratio[i].bExecute := TRUE;
		END_FOR
		StateNext(state_main);
	19:// set gear done
		axiss_ready_all := TRUE;
		FOR i := 0 TO c_axis_i_max BY 1 DO
			axiss_ready_all := axiss_ready_all AND axiss_change_gearing_ratio[i].bDone AND NOT axiss_change_gearing_ratio[i].bError;
		END_FOR
		IF axiss_ready_all THEN
			FOR i := 0 TO c_axis_i_max BY 1 DO
				axiss_change_gearing_ratio[i].bExecute := FALSE;
			END_FOR
			StateNext(state_main);
		END_IF
	20:// reinit drive
		FOR i := 0 TO c_axis_i_max BY 1 DO
			axiss_reinit_drive[i].bExecute := TRUE;
		END_FOR
		StateNext(state_main);
	21:// reinit drive done
		axiss_ready_all := TRUE;
		FOR i := 0 TO c_axis_i_max BY 1 DO
			axiss_ready_all := axiss_ready_all AND axiss_reinit_drive[i].bDone AND axiss[i]^.wCommunicationState = 100;
		END_FOR
		IF axiss_ready_all THEN
			FOR i := 0 TO c_axis_i_max BY 1 DO
				axiss_reinit_drive[i].bExecute := FALSE;
			END_FOR
			StateNext(state_main);
		END_IF
	22:// calculate max
		FOR i := 0 TO c_axis_i_max BY 1 DO
			axiss_max_μ_per_sec[i] := (axiss_encoder_resolution[i] * (MIN(axiss_max_rpm[i], save.max_rpm[i]) / 60)) / ABS(axiss[i]^.fScalefactor);
		END_FOR
		StateNext(state_main);
	23:// prepair
		FOR i := 0 TO c_axis_i_max BY 1 DO
			axiss_power[i].Enable := TRUE;
			axiss_power[i].bRegulatorOn := TRUE;
		END_FOR
		StateNext(state_main);
	24:
		save_apply();
		StateNext(state_main);
	25:
		hmi.plc_ready := TRUE; // sau khi đã khởi động Servo bla bla thì ta PLC ready
		work_data.state := State.RST; // reset work
		state_main := State.RUN_ING; // bước vào giai đoạn chạy
		supply_fb.d := ADR(supply_data);
		tap_fb.d := ADR(tap_data);
	State.RUN_ING:
		io(); // kiểm tra io (gồm PLC io và HMI)
		supply_fb(d:= );
		tap_fb(d:= );
		work();
END_CASE

ACTION io:
////////////
//HMI DOWN//
///////////
IF hmi.hmi_ready THEN
	////////
	//WORK//
	////////
	// basis
	work_data.input_run.rise(CLK:= hmi.run, Q=> );
	work_data.input_stop.rise(CLK:= hmi.stop, Q=> );
	work_data.input_home.rise(CLK:= hmi.home, Q=> );
	// test
	work_data.supply_test.timer(IN:= hmi.supply_test, PT:= , Q=> , ET=> );
	// fix problem
	supply_data.no_air.fix_rise(CLK:= hmi.problem_fix[0], Q=> );
	work_data.overload.fix_rise(CLK:= hmi.problem_fix[1], Q=> );
	supply_data.foil_stuck.fix_rise(CLK:= hmi.problem_fix[2], Q=> );
	////////
	//SAVE//
	////////
	IF hmi.sv_need_check THEN
		save_check();
		hmi.sv_need_check := FALSE;
	END_IF
	main_save.rise(CLK:= hmi.sv_trigger, Q=> ); // Trên HMI sẽ xuất hiện nút save khi biến hmi_data.save_need = true.
	IF main_save.rise.Q THEN
		save := hmi.sv;
		save_apply();
		hmi.sv_need := FALSE;
		hmi.sv_trigger := FALSE;
	END_IF
END_IF
/////////
//INPUT//
/////////
supply_data.axis.encoder_single_position := DWORD_TO_DINT(%ID5);
tap_data.axis_move.encoder_single_position := DWORD_TO_DINT(%ID10);
tap_data.axis_spin.encoder_single_position := DWORD_TO_DINT(%ID15);
tap_data.time_delta_sec := time_delta_sec;
//
IF NOT test THEN
	work_data.input_run.rise_physical.CLK := %IX0.0;
	work_data.input_stop.fall_physical.CLK := %IX0.1;
	supply_data.input_air := %IX0.2;
	supply_data.input_foil := %IX0.3;
END_IF
// delay các xylanh
supply_data.clamp.n_timer(IN:= NOT supply_data.clamp.on, PT:= , Q=> , ET=> );
supply_data.clamp.p_timer(IN:= supply_data.clamp.on, PT:= , Q=> , ET=> );
supply_data.extract_down.n_timer(IN:= NOT supply_data.extract_down.on, PT:= , Q=> , ET=> );
supply_data.extract_down.p_timer(IN:= supply_data.extract_down.on, PT:= , Q=> , ET=> );
supply_data.extract_pull.n_timer(IN:= NOT supply_data.extract_pull.on, PT:= , Q=> , ET=> );
supply_data.extract_pull.p_timer(IN:= supply_data.extract_pull.on, PT:= , Q=> , ET=> );
// điều kiện thực hiện các lệnh
work_data.can_run := work_data.input_stop.fall_physical.CLK AND supply_data.input_air AND work_data.state = State.READY;
work_data.can_stop := work_data.state >= State.NONE;
work_data.can_home := work_data.state = State.RST_DONE OR work_data.state = State.READY;
// xảy ra lỗi
supply_data.no_air.rise(CLK:= NOT supply_data.input_air, Q=> );
IF supply_data.no_air.rise.Q THEN
	supply_data.no_air.on := TRUE;
END_IF
IF supply_data.axis.overload OR tap_data.axis_move.overload OR tap_data.axis_spin.overload OR tap_data.deviation_overload THEN
	work_data.overload.on := TRUE;
END_IF
work_data.overload.rise(CLK:= work_data.overload.on, Q=> );
IF (work_data.input_stop.rise.Q OR work_data.input_stop.fall_physical.Q OR supply_data.no_air.rise.Q OR work_data.overload.rise.Q) AND work_data.can_stop THEN
	hmi.jog_micro_per_sec_or_rev := 0;
	work_data.auto.on := FALSE;
	work_data.state := State.RST;
END_IF
supply_data.foil_stuck.rise(CLK:= supply_data.foil_stuck.timer.Q, Q=> );
IF supply_data.foil_stuck.rise.Q THEN
	supply_data.foil_stuck.on := TRUE;
END_IF
// nhấn sửa lỗi xong
IF supply_data.no_air.fix_rise.Q AND supply_data.input_air THEN
	supply_data.no_air.on := FALSE;
END_IF
IF work_data.overload.fix_rise.Q THEN
	supply_data.axis.overload := FALSE;
	tap_data.axis_move.overload := FALSE;
	tap_data.axis_spin.overload := FALSE;
	tap_data.deviation_overload := FALSE;
	supply_data.axis.overload_hold_torque_timer.IN := FALSE;
	tap_data.axis_move.overload_hold_torque_timer.IN := FALSE;
	tap_data.axis_spin.overload_hold_torque_timer.IN := FALSE;
	work_data.overload.on := FALSE;
END_IF
IF supply_data.foil_stuck.fix_rise.Q THEN
	supply_data.foil_stuck.on := FALSE;
	supply_data.foil_stuck.timer.IN := FALSE;
END_IF
// thao tác chạy máy
work_data.input_run.rise_physical(CLK:= , Q=> );
work_data.input_stop.fall_physical(CLK:= , Q=> );
work_data.input_run.timer(IN:= work_data.input_run.rise.CLK OR work_data.input_run.rise_physical.CLK, PT:= , Q=> , ET=> );
work_data.auto.timer(IN:= work_data.input_run.rise.CLK OR work_data.input_run.rise_physical.CLK, PT:= , Q=> , ET=> );
IF work_data.input_home.rise.Q AND work_data.can_home THEN
	supply_data.axis.home_done := FALSE;
	tap_data.axis_move.home_done := FALSE;
	tap_data.axis_spin.home_done := FALSE;
	work_data.state := State.HOME;
END_IF
IF work_data.input_stop.fall_physical.CLK AND NOT supply_data.no_air.on AND NOT work_data.overload.on THEN
	IF work_data.auto.timer.Q THEN
		work_data.auto.on := TRUE;
	END_IF
	CASE work_data.state OF
		State.RST_DONE:
			IF work_data.input_run.rise.Q OR work_data.input_run.rise_physical.Q THEN
				work_data.state := State.HOME;
			END_IF
		State.READY:
			IF work_data.can_run AND supply_data.state = State.READY AND tap_data.state = State.READY THEN
				IF work_data.input_run.timer.Q OR work_data.auto.on THEN
					work_data.state := State.RUN;
				END_IF
			END_IF
		ELSE
			IF work_data.auto.on AND (work_data.input_run.rise.Q OR work_data.input_run.rise_physical.Q) THEN
				work_data.auto.on := FALSE;
			END_IF
	END_CASE
END_IF
// thao tác thử máy
work_data.supply_test.rise(CLK:= work_data.supply_test.timer.Q, Q=> );
IF supply_data.input_air AND work_data.manual THEN
	IF supply_data.state = State.READY THEN
		supply_data.clamp.on := hmi.supply_clamp;
		supply_data.extract_down.on := hmi.supply_extract_down;
		supply_data.extract_pull.on := hmi.supply_extract_pull;
		IF NOT tap_data.lubricate.on THEN
			tap_data.lubricate.on := hmi.tap_lubricate;
		END_IF
		IF NOT supply_data.clean.on THEN
			supply_data.clean.on := hmi.supply_clean;
		END_IF
		IF work_data.supply_test.rise.Q THEN
			supply_data.state := 111;
		END_IF
	ELSE
		hmi.supply_clamp := supply_data.clamp.on;
		hmi.tap_lubricate := tap_data.lubricate.on;
		hmi.supply_clean := supply_data.clean.on;
	END_IF
ELSE
	hmi.supply_clamp := supply_data.clamp.on;
	hmi.supply_extract_down := supply_data.extract_down.on;
	hmi.supply_extract_pull := supply_data.extract_pull.on;
	hmi.tap_lubricate := tap_data.lubricate.on;
	hmi.supply_clean := supply_data.clean.on;
END_IF
//////////
//OUTPUT//
//////////
work_data.alarm := supply_data.no_air.on OR work_data.overload.on;
%QX0.0 := supply_data.clamp.on; // kẹp phôi
%QX0.1 := tap_data.lubricate.on; // bôi trơn
%QX0.2 := supply_data.clean.on; // làm sạch + đẩy phôi vào mâm
%QX0.3 := work_data.alarm; // lỗi
tap_data.lubricate.timer(IN:= tap_data.lubricate.on, PT:= , Q=> , ET=> );
IF tap_data.lubricate.timer.Q THEN
	tap_data.lubricate.on := FALSE;
	hmi.tap_lubricate := FALSE;
END_IF
supply_data.clean.timer(IN:= supply_data.clean.on, PT:= , Q=> , ET=> );
IF supply_data.clean.timer.Q THEN
	supply_data.clean.on := FALSE;
	hmi.supply_clean := FALSE;
END_IF
//////////
//HMI UP//
//////////
IF hmi.hmi_ready THEN
	hmi.view_input[0] := work_data.input_run.rise_physical.CLK;
	hmi.view_input[1] := work_data.input_stop.fall_physical.CLK;
	hmi.view_input[2] := supply_data.input_air;
	hmi.view_input[3] := supply_data.input_foil;
	//
	hmi.view_output[0] := supply_data.clamp.on;
	hmi.view_output[1] := tap_data.lubricate.on;
	hmi.view_output[2] := supply_data.clean.on;
	hmi.view_output[3] := work_data.alarm;
	//
	hmi.view_can_run := work_data.can_run;
	hmi.view_can_stop := work_data.can_stop;
	hmi.view_can_home := work_data.can_home;
	hmi.view_auto := work_data.auto.on;
	hmi.view_manual := work_data.manual;
	//
	hmi.view_problem[0] := supply_data.no_air.on;
	hmi.view_problem[1] := work_data.overload.on;
	hmi.view_problem[2] := supply_data.foil_stuck.on;
	//
	hmi.view_tap_deviation_micron := LREAL_TO_UINT(tap_data.deviation_μm);
	hmi.view_cycle_count := cycle_count;
	hmi.view_cycle_time_msec := work_data.cycle_time_msec;
	//
	hmi.view_axis_encoder[0] := supply_data.axis.encoder_single_position;
	hmi.view_axis_encoder[1] := tap_data.axis_move.encoder_single_position;
	hmi.view_axis_encoder[2] := tap_data.axis_spin.encoder_single_position;
	hmi.view_axis_micro[0] := LREAL_TO_DINT(supply_data.axis.ref^.fActPosition);
	hmi.view_axis_micro[1] := LREAL_TO_DINT(tap_data.axis_move.ref^.fActPosition);
	hmi.view_axis_micro[2] := LREAL_TO_DINT(tap_data.axis_spin.ref^.fActPosition);
	hmi.view_axis_mNm[0] := LREAL_TO_UDINT(supply_data.axis.torque_Nm_abs * 1E3);
	hmi.view_axis_mNm[1] := LREAL_TO_UDINT(tap_data.axis_move.torque_Nm_abs * 1E3);
	hmi.view_axis_mNm[2] := LREAL_TO_UDINT(tap_data.axis_spin.torque_Nm_abs * 1E3);
	//
	hmi.view_load := LREAL_TO_UINT(tap_data.load * 1E3);
	//
	hmi.view_state[1] := work_data.state;
	hmi.view_state[2] := supply_data.state;
	hmi.view_state[3] := tap_data.state;
END_IF
END_ACTION

ACTION motion:
FOR i := 0 TO c_axis_i_max BY 1 DO
	axiss_read[i](
		xExecute:= , 
		xAbort:= , 
		uiIndex:= , 
		usiSubIndex:= , 
		Axis:= axiss[i]^, 
		xDone=> , 
		xBusy=> , 
		xError=> , 
		usiDataLength=> , 
		dwValue=> , 
		dwErrorCode=> , 
		eError=> );
	axiss_write[i](
		xExecute:= , 
		xAbort:= , 
		uiIndex:= , 
		usiSubIndex:= , 
		usiDataLength:= , 
		dwValue:= , 
		Axis:= axiss[i]^, 
		xDone=> , 
		xBusy=> , 
		xError=> , 
		dwErrorCode=> , 
		eError=> );
	axiss_read_status[i](
		Axis:= axiss[i]^, 
		Enable:= , 
		Valid=> , 
		Busy=> , 
		Error=> , 
		ErrorID=> , 
		Disabled=> , 
		Errorstop=> , 
		Stopping=> , 
		StandStill=> , 
		DiscreteMotion=> , 
		ContinuousMotion=> , 
		SynchronizedMotion=> , 
		Homing=> , 
		ConstantVelocity=> , 
		Accelerating=> , 
		Decelerating=> , 
		FBErrorOccured=> );
	axiss_change_gearing_ratio[i](
		Axis:= axiss[i]^, 
		bExecute:= , 
		dwRatioTechUnitsDenom:= , 
		iRatioTechUnitsNum:= , 
		fPositionPeriod:= , 
		iMovementType:= , 
		bDone=> , 
		bBusy=> , 
		bError=> , 
		nErrorID=> );
	axiss_reinit_drive[i](
		Axis:= axiss[i]^, 
		bExecute:= , 
		bVirtual:= , 
		bDone=> , 
		bBusy=> , 
		bError=> , 
		nErrorID=> );
	axiss_set_mode[i](
		Axis:= axiss[i]^, 
		bExecute:= , 
		nControllerMode:= , 
		bDone=> , 
		bBusy=> , 
		bError=> , 
		nErrorID=> );
	axiss_power[i](
		Axis:= axiss[i]^,
		Enable:= , 
		bRegulatorOn:= , 
		bDriveStart:= , 
		Status=> , 
		bRegulatorRealState=> , 
		bDriveStartRealState=> , 
		Busy=> , 
		Error=> , 
		ErrorID=> );
	axiss_reset[i](
		Axis:= axiss[i]^,
		Execute:= ,
		Done=> ,
		Busy=> ,
		Error=> ,
		ErrorID=> );
	axiss_stop[i](
		Axis:= axiss[i]^, 
		Execute:= , 
		Deceleration:= , 
		Jerk:= , 
		Done=> , 
		Busy=> , 
		Error=> , 
		ErrorID=> );
	axiss_inch[i](
		Axis:= axiss[i]^, 
		InchForward:= , 
		InchBackward:= , 
		Distance:= , 
		Velocity:= , 
		Acceleration:= , 
		Deceleration:= , 
		Jerk:= , 
		Busy=> , 
		CommandAborted=> , 
		Error=> , 
		ErrorId=> );
	axiss_fsv[i](
		Axis:= axiss[i]^, 
		bExecute:= , 
		bAbort:= , 
		dwValueMask:= , 
		fSetPosition:= , 
		fSetVelocity:= , 
		fSetAcceleration:= , 
		fSetJerk:= , 
		fSetTorque:= , 
		fSetCurrent:= , 
		bBusy=> , 
		bCommandAborted=> , 
		bError=> , 
		iErrorID=> );
	axiss_sp[i](
		Axis:= axiss[i]^, 
		Execute:= , 
		Position:= , 
		Mode:= , 
		Done=> , 
		Busy=> , 
		Error=> , 
		ErrorID=> );
	axiss_mabs[i](
		Axis:= axiss[i]^, 
		Execute:= , 
		Position:= , 
		Velocity:= , 
		Acceleration:= , 
		Deceleration:= , 
		Jerk:= , 
		Direction:= , 
		BufferMode:= , 
		Done=> , 
		Busy=> , 
		Active=> , 
		CommandAborted=> , 
		Error=> , 
		ErrorID=> );
END_FOR
END_ACTION

ACTION save_check:
hmi.sv_need := (
	save.home_encoder_value_recorded <> hmi.sv.home_encoder_value_recorded OR
	save.max_micro_recorded <> hmi.sv.max_micro_recorded OR
	//
	save.supply_micro_per_sec <> hmi.sv.supply_micro_per_sec OR
	//
	save.tap_begin_micron <> hmi.sv.tap_begin_micron OR
	save.tap_depth_micron <> hmi.sv.tap_depth_micron OR
	save.tap_micron_per_rev <> hmi.sv.tap_micron_per_rev OR
	save.tap_rpm <> hmi.sv.tap_rpm OR
	save.tap_backlash_micro <> hmi.sv.tap_backlash_micro OR
	save.tap_deviation_micron_max <> hmi.sv.tap_deviation_micron_max
);
FOR i := 0 TO c_cylinder_i_max BY 1 DO
	hmi.sv_need := (hmi.sv_need OR
		save.cylinder_n_delay_msec[i] <> hmi.sv.cylinder_n_delay_msec[i] OR
		save.cylinder_p_delay_msec[i] <> hmi.sv.cylinder_p_delay_msec[i]
	);
END_FOR
FOR i := 0 TO c_air_burst_i_max BY 1 DO
	hmi.sv_need := (hmi.sv_need OR
		save.air_burst_delay_msec[i] <> hmi.sv.air_burst_delay_msec[i]
	);
END_FOR
FOR i := 0 TO c_axis_i_max BY 1 DO
	hmi.sv_need := (hmi.sv_need OR
		save.max_rpm[i] <> hmi.sv.max_rpm[i] OR
		save.gear_dir[i] <> hmi.sv.gear_dir[i] OR
		save.gear_num[i] <> hmi.sv.gear_num[i] OR
		save.gear_den[i] <> hmi.sv.gear_den[i] OR
		save.home_torque_mNm[i] <> hmi.sv.home_torque_mNm[i] OR
		save.home_encoder_value[i] <> hmi.sv.home_encoder_value[i] OR
		save.max_micro[i] <> hmi.sv.max_micro[i] OR
		save.overload_hold_torque_factor[i] <> hmi.sv.overload_hold_torque_factor[i] OR
		save.overload_hold_torque_time_msec[i] <> hmi.sv.overload_hold_torque_time_msec[i] OR
		save.overload_instant_torque_factor[i] <> hmi.sv.overload_instant_torque_factor[i] OR
		save.ramp_time_msec[i] <> hmi.sv.ramp_time_msec[i] OR
		save.jerk_factor[i] <> hmi.sv.jerk_factor[i]
	);
END_FOR
END_ACTION

ACTION save_apply:
/////////
//LIMIT//
/////////
FOR i := 0 TO c_cylinder_i_max DO
	save.cylinder_n_delay_msec[i] := MAX(0_100, MIN(5_000, save.cylinder_n_delay_msec[i]));
	save.cylinder_p_delay_msec[i] := MAX(0_100, MIN(5_000, save.cylinder_p_delay_msec[i]));
END_FOR
FOR i := 0 TO c_air_burst_i_max DO
	save.air_burst_delay_msec[i] := MAX(0_100, MIN(5_000, save.air_burst_delay_msec[i]));
END_FOR
FOR i := 0 TO c_axis_i_max BY 1 DO
	save.max_rpm[i] := MAX(1000, MIN(axiss_max_rpm[i] - 200, save.max_rpm[i]));
	save.gear_num[i] := MAX(1, save.gear_num[i]);
	save.gear_den[i] := MAX(1, save.gear_den[i]);
	save.home_torque_mNm[i] := MAX(0_100, MIN(LREAL_TO_UINT(axiss_rated_torque_Nm[i] * 1E3), save.home_torque_mNm[i]));
	save.home_encoder_value[i] := MAX(0, MIN(axiss_encoder_resolution[i] - 1, save.home_encoder_value[i]));
	save.max_micro[i] := MAX(10_000, save.max_micro[i]);
	save.overload_hold_torque_factor[i] := MAX(0_010, MIN(3_000, save.overload_hold_torque_factor[i]));
	save.overload_hold_torque_time_msec[i] := MAX(0_010, MIN(2_000, save.overload_hold_torque_time_msec[i]));
	save.overload_instant_torque_factor[i] := MAX(0_010, MIN(3_000, save.overload_instant_torque_factor[i]));
	save.ramp_time_msec[i] := MAX(0_050, MIN(0_800, save.ramp_time_msec[i]));
	save.jerk_factor[i] := MAX(5, MIN(80, save.jerk_factor[i]));
END_FOR
//
save.supply_micro_per_sec := MAX(0_100, MIN(LREAL_TO_UDINT(axiss_max_μ_per_sec[0]), save.supply_micro_per_sec));
//
save.tap_begin_micron := MAX(1_000, MIN(DINT_TO_UDINT(save.max_micro[2]) - 1_000, save.tap_begin_micron));
save.tap_depth_micron := MAX(1_000, MIN(DINT_TO_UDINT(save.max_micro[2]) - save.tap_begin_micron, save.tap_depth_micron));
save.tap_micron_per_rev := MAX(0_500, MIN(2_000, save.tap_micron_per_rev));
save.tap_rpm := MAX(100, MIN(save.max_rpm[2], save.tap_rpm));
save.tap_backlash_micro := MIN(1_000, save.tap_backlash_micro);
save.tap_deviation_micron_max := MAX(0_001, save.tap_deviation_micron_max);
/////////
//APPLY//
/////////
FOR i := 0 TO c_axis_i_max BY 1 DO
	CASE i OF
		0: axis_ec_i := ADR(supply_data.axis);
		1: axis_ec_i := ADR(tap_data.axis_move);
		2: axis_ec_i := ADR(tap_data.axis_spin);
	END_CASE
	axis_ec_i^.home_encoder_value_recorded := save.home_encoder_value_recorded;
	axis_ec_i^.home_encoder_value_save := ADR(save.home_encoder_value[i]);
	axis_ec_i^.max_μ_recorded := save.max_micro_recorded;
	axis_ec_i^.max_μ_save := ADR(save.max_micro[i]);
	axis_ec_i^.max_μ := DINT_TO_LREAL(axis_ec_i^.max_μ_save^);
	axis_ec_i^.max_μ_per_sec := axiss_max_μ_per_sec[i];
	axis_ec_i^.home_torque_Nm := UINT_TO_LREAL(save.home_torque_mNm[i]) * 1E-3;
	axis_ec_i^.home_hit_timer.PT := INT_TO_TIME(1_000);
	axis_ec_i^.home_offset_absolute_μ := 5_000;
	axis_ec_i^.home_back_μ_per_sec := MIN(10_000, axis_ec_i^.max_μ_per_sec);
	axis_ec_i^.home_forward_μ_per_sec := MIN(30_000, axis_ec_i^.max_μ_per_sec);
	axis_ec_i^.overload_hold_torque_Nm := axis_ec_i^.torque_rated_Nm * save.overload_hold_torque_factor[i] * 1E-3;
	axis_ec_i^.overload_hold_torque_timer.PT := UINT_TO_TIME(save.overload_hold_torque_time_msec[i]);
	axis_ec_i^.overload_instant_torque_Nm := axis_ec_i^.torque_rated_Nm * save.overload_instant_torque_factor[i] * 1E-3;
	axis_ec_i^.ramp_time_sec := UINT_TO_LREAL(save.ramp_time_msec[i]) * 1E-3;
	axis_ec_i^.jerk_factor := save.jerk_factor[i];
END_FOR
supply_data.axis.max_μ := 1E16;
//
FOR i := 0 TO c_cylinder_i_max DO
	CASE i OF
		0: cylinder_i := ADR(supply_data.clamp);
		1: cylinder_i := ADR(supply_data.extract_down);
		2: cylinder_i := ADR(supply_data.extract_pull);
	END_CASE
	cylinder_i^.n_timer.PT := UINT_TO_TIME(save.cylinder_n_delay_msec[i]);
	cylinder_i^.p_timer.PT := UINT_TO_TIME(save.cylinder_p_delay_msec[i]);
END_FOR
FOR i := 0 TO c_air_burst_i_max DO
	CASE i OF
		0: air_burst_i := ADR(tap_data.lubricate);
		1: air_burst_i := ADR(supply_data.clean);
	END_CASE
	air_burst_i^.timer.PT := UINT_TO_TIME(save.air_burst_delay_msec[i]);
END_FOR
//tap
tap_data.begin_μm := UDINT_TO_LREAL(save.tap_begin_micron);
tap_data.depth_μm := UDINT_TO_LREAL(save.tap_depth_micron);
tap_data.μm_per_rev := UDINT_TO_LREAL(save.tap_micron_per_rev);
tap_data.rps := UDINT_TO_LREAL(save.tap_rpm) / 60;
tap_data.backlash_μ := UINT_TO_LREAL(save.tap_backlash_micro);
tap_data.deviation_μm_max := UINT_TO_LREAL(save.tap_deviation_micron_max);
//
supply_data.μ_per_sec := save.supply_micro_per_sec;
supply_data.foil_stuck.timer.PT := INT_TO_TIME(1_000);
//
work_data.input_run.timer.PT := INT_TO_TIME(0_300);
work_data.auto.timer.PT := INT_TO_TIME(2_000);
work_data.supply_test.timer.PT := INT_TO_TIME(0_300);
/////////
//FINAL//
/////////
hmi.sv := save;
END_ACTION

ACTION work:
CASE work_data.state OF
	State.RST:
		work_data.manual := FALSE;
		work_data.alarm := FALSE;
		tap_data.state := State.RST;
		StateNext(work_data.state);
	2:
		IF tap_data.state = State.RST_DONE THEN
			supply_data.state_extract := State.RST;
			StateNext(work_data.state);
		END_IF
	3:
		IF supply_data.state_extract = State.READY THEN
			supply_data.state := State.RST;
			StateNext(work_data.state);
		END_IF
	4:
		IF supply_data.state = State.RST_DONE THEN
			work_data.state := State.RST_DONE;
		END_IF
	State.RST_DONE:
		//do nothing
	//////\\
	////\\\\
	//\\\\\\
	State.HOME:
		tap_data.state := State.HOME;
		StateNext(work_data.state);
	52:
		IF tap_data.state = State.HOME_DONE THEN
			supply_data.state := State.HOME;
			StateNext(work_data.state);
		END_IF
	53:
		IF supply_data.state = State.HOME_DONE THEN
			work_data.state := State.HOME_DONE;
		END_IF
	//
	State.HOME_DONE:
		supply_data.state := State.HOME_OFFSET;
		tap_data.state := State.HOME_OFFSET;
		StateNext(work_data.state);
	91:
		IF (
			supply_data.state = State.HOME_OFFSET_DONE AND
			tap_data.state = State.HOME_OFFSET_DONE
		) THEN
			work_data.state := State.HOME_OFFSET_DONE;
		END_IF
	State.HOME_OFFSET_DONE:
		supply_data.state := State.READY;
		supply_data.state_extract := State.READY;
		tap_data.state := State.READY;
		work_data.state := State.READY;
		work_data.manual := TRUE;
		IF NOT save.home_encoder_value_recorded THEN
			save.home_encoder_value_recorded := TRUE;
			save.max_micro_recorded := TRUE;
			save_apply();
		END_IF
	//////\\
	////\\\\
	//\\\\\\
	State.READY:
		IF work_data.manual THEN
			tap_data.axis_v_inch.InchBackward := hmi.jog_n;
			tap_data.axis_v_inch.InchForward := hmi.jog_p;
			tap_data.axis_v_inch.Velocity := hmi.jog_micro_per_sec_or_rev;
			tap_data.axis_v_inch.Acceleration := tap_data.axis_v_inch.Velocity / tap_data.axis_move.ramp_time_sec;
			tap_data.axis_v_inch.Deceleration := tap_data.axis_v_inch.Acceleration;
			tap_data.axis_v_inch.Jerk := tap_data.axis_v_inch.Acceleration * tap_data.axis_move.jerk_factor;
			IF hmi.jog_n THEN
				tap_data.axis_v_inch.Distance := tap_data.axis_v^.fActPosition;
			END_IF
			IF hmi.jog_p THEN
				tap_data.axis_v_inch.Distance := tap_data.axis_move.max_μ - tap_data.axis_v^.fActPosition;
			END_IF
		END_IF
	//////\\
	////\\\\
	//\\\\\\
	State.RUN:
		work_data.manual := FALSE;
		supply_data.clamp.on := TRUE;
		work_data.cycle_start_msec := time_msec;
		StateNext(work_data.state);
	102:
		IF supply_data.clamp.p_timer.Q THEN
			tap_data.state := State.RUN;
			supply_data.state_extract := State.RUN;
			StateNext(work_data.state);
		END_IF
	103:
		IF tap_data.state = State.READY AND supply_data.state_extract = State.READY THEN
			supply_data.state := State.RUN;
			StateNext(work_data.state);
		END_IF
	104:
		IF supply_data.state = State.READY THEN
			work_data.state := 131;
		END_IF
	//end
	131:
		work_data.state := State.READY;
		work_data.cycle_time_msec := ULINT_TO_UDINT(time_msec - work_data.cycle_start_msec);
		work_data.alarm := FALSE;
		IF (time_msec - cycle_count_reset_time_msec) > 86400_000 THEN
			cycle_count := 0;
			cycle_count_reset_time_msec := (time_msec / 86400_000) * 86400_000;
		END_IF
		cycle_count := cycle_count + 1;
END_CASE
END_ACTION

END_PROGRAM

// Device/Application/StateNext
FUNCTION StateNext
VAR_INPUT
	state: REFERENCE TO INT;
END_VAR
VAR
END_VAR

state := state + 1;

END_FUNCTION

// Device/Application/SupplyFB
FUNCTION_BLOCK SupplyFB
VAR_INPUT
	d: POINTER TO SupplyData;
END_VAR

////////
//MAIN//
////////
d^.axis_fb(d:= ); // data của hàm này đã được set ở hàm MAIN
d^.foil_stuck.timer(IN:= , PT:= , Q=> , ET=> );
CASE d^.state OF
	//////\\
	////\\\\
	//\\\\\\
	State.RST:
		d^.axis.overload_check := FALSE;
		d^.clamp.on := FALSE;
		d^.foil_stuck.timer.IN := FALSE;
		StateNext(d^.state);
	2:
		IF d^.clamp.n_timer.Q THEN
			d^.axis.state := State.RST;
			StateNext(d^.state);
		END_IF
	3:
		IF d^.axis.state = State.RST_DONE THEN
			d^.state := State.RST_DONE;
		END_IF
	//////\\
	////\\\\
	//\\\\\\
	State.HOME:
		d^.clamp.on := FALSE;
		StateNext(d^.state);
	52:
		IF d^.clamp.n_timer.Q THEN
			d^.axis.home_to_encoder := TRUE;
			d^.axis.home_encoder_value_recorded := TRUE;
			d^.axis.home_done_forward_ignore := TRUE;
			d^.axis.state := State.HOME;
			StateNext(d^.state);
		END_IF
	53:
		IF d^.axis.state = State.HOME_DONE THEN
			d^.axis.overload_check := TRUE;
			d^.state := State.HOME_DONE;
		END_IF
	//////\\
	////\\\\
	//\\\\\\
	State.HOME_OFFSET:
		d^.axis.home_offset_μ := 0;
		d^.axis.state := State.HOME_OFFSET;
		StateNext(d^.state);
	92:
		IF d^.axis.state = State.HOME_OFFSET_DONE THEN
			d^.axis.state := State.READY;
			d^.state := State.HOME_OFFSET_DONE;
		END_IF
	State.READY:
		//do nothing
	//////\\
	////\\\\
	//\\\\\\
	State.RUN:
		d^.clamp.on := FALSE;
		d^.foil_stuck.timer.IN := TRUE;
		StateNext(d^.state);
	102:
		IF d^.input_foil AND NOT d^.foil_stuck.on THEN
			d^.foil_stuck.timer.IN := FALSE;
			StateNext(d^.state);
		END_IF
	103:
		IF (
			d^.clamp.n_timer.Q AND
			d^.axis.state = State.READY
		) THEN
			d^.axis.target_position_μ := 1_000; // trục module 1000, nên vị trí luôn < 1000, chạy tới vị trí 1000 sẽ quay 1 vòng
			d^.axis.target_velocity_μ_per_sec := d^.μ_per_sec;
			d^.axis.mabs^.Direction := MC_DIRECTION.positive;
			d^.axis.state := State.RUN;
			StateNext(d^.state);
		END_IF
	104:
		IF d^.axis.state = State.READY THEN
			d^.clean.on := TRUE;
			d^.state := State.READY;
		END_IF
	//////\\
	////\\\\
	//\\\\\\
	111: // supply test
		d^.clamp.on := FALSE;
		d^.state_extract := State.RST;
		StateNext(d^.state);
	112:
		IF (
			d^.clamp.n_timer.Q AND
			d^.state_extract = State.READY AND
			d^.axis.state = State.READY
		) THEN
			d^.axis.target_position_μ := 1_000;
			d^.axis.target_velocity_μ_per_sec := d^.μ_per_sec;
			d^.axis.mabs^.Direction := MC_DIRECTION.positive;
			d^.axis.state := State.RUN;
			StateNext(d^.state);
		END_IF
	113:
		IF d^.axis.state = State.READY THEN
			d^.state := State.READY;
		END_IF
END_CASE
///////////
//EXTRACT//
///////////
CASE d^.state_extract OF
	State.RST:
		d^.extract_down.on := FALSE;
		d^.extract_pull.on := FALSE;
		StateNext(d^.state_extract);
	2:
		IF (
			d^.extract_down.n_timer.Q AND
			d^.extract_pull.n_timer.Q
		) THEN
			d^.state_extract := State.READY;
		END_IF
	//////\\
	////\\\\
	//\\\\\\
	State.RUN:
		d^.extract_pull.on := TRUE;
		StateNext(d^.state_extract);
	102:
		IF d^.extract_pull.p_timer.Q THEN
			d^.extract_down.on := TRUE;
			StateNext(d^.state_extract);
		END_IF
	103:
		IF d^.extract_down.p_timer.Q THEN
			d^.extract_pull.on := FALSE;
			StateNext(d^.state_extract);
		END_IF
	104:
		IF d^.extract_pull.n_timer.Q THEN
			d^.extract_down.on := FALSE;
			StateNext(d^.state_extract);
		END_IF
	105:
		IF d^.extract_down.n_timer.Q THEN
			d^.state_extract := State.READY;
		END_IF
END_CASE

END_FUNCTION_BLOCK

// Device/Application/TapFB
FUNCTION_BLOCK TapFB
VAR_INPUT
	d: POINTER TO TapData;
END_VAR

////////
//MAIN//
////////
d^.axis_move_fb(d:= ); // data của hàm này đã được set ở hàm MAIN
d^.axis_spin_fb(d:= );
d^.axis_v_power(
	Axis:= d^.axis_v^, 
	Enable:= , 
	bRegulatorOn:= , 
	bDriveStart:= , 
	Status=> , 
	bRegulatorRealState=> , 
	bDriveStartRealState=> , 
	Busy=> , 
	Error=> , 
	ErrorID=> );
d^.axis_v_stop(
	Axis:= d^.axis_v^, 
	Execute:= , 
	Deceleration:= , 
	Jerk:= , 
	Done=> , 
	Busy=> , 
	Error=> , 
	ErrorID=> );
d^.axis_v_inch(
	Axis:= d^.axis_v^, 
	InchForward:= , 
	InchBackward:= , 
	Distance:= , 
	Velocity:= , 
	Acceleration:= , 
	Deceleration:= , 
	Jerk:= , 
	Busy=> , 
	CommandAborted=> , 
	Error=> , 
	ErrorId=> );
d^.axis_v_sp(
	Axis:= d^.axis_v^, 
	Execute:= , 
	Position:= , 
	Mode:= , 
	Done=> , 
	Busy=> , 
	Error=> , 
	ErrorID=> );
d^.axis_v_mabs(
	Axis:= d^.axis_v^, 
	Execute:= , 
	Position:= , 
	Velocity:= , 
	Acceleration:= , 
	Deceleration:= , 
	Jerk:= , 
	Direction:= , 
	BufferMode:= , 
	Done=> , 
	Busy=> , 
	Active=> , 
	CommandAborted=> , 
	Error=> , 
	ErrorID=> );
IF d^.axis_move.overload_check AND d^.axis_spin.overload_check AND (d^.state = State.READY OR d^.state = 105) THEN
	d^.deviation_μm := ABS(d^.axis_move_follow_data.deviation - d^.axis_spin_follow_data.deviation);
	IF d^.deviation_μm >= d^.deviation_μm_max THEN
		d^.deviation_overload := TRUE;
	END_IF
END_IF
CASE d^.state OF
	//////\\
	////\\\\
	//\\\\\\
	State.RST:
		d^.axis_move.overload_check := FALSE;
		d^.axis_spin.overload_check := FALSE;
		d^.axis_move.jog_type := JogType.FSV;
		d^.axis_spin.jog_type := JogType.FSV;
		d^.axis_v_inch.InchBackward := FALSE;
		d^.axis_v_inch.InchForward := FALSE;
		d^.axis_move.state := State.RST;
		d^.axis_spin.state := State.RST;
		StateNext(d^.state);
	2:
		IF (
			d^.axis_move.state = State.RST_DONE AND
			d^.axis_spin.state = State.RST_DONE
		) THEN
			StateNext(d^.state);
		END_IF
	3:
		d^.axis_v_power.Enable := TRUE;
		d^.axis_v_power.bRegulatorOn := TRUE;
		d^.axis_v_power.bDriveStart := TRUE;
		StateNext(d^.state);
	4:
		IF d^.axis_v_power.Status THEN
			StateNext(d^.state);
		END_IF
	5:
		IF d^.axis_v_mabs.Busy THEN
			d^.axis_v_stop.Deceleration := d^.rps * d^.μm_per_rev / d^.axis_move.ramp_time_sec;
			d^.axis_v_stop.Jerk := d^.axis_v_stop.Deceleration * d^.axis_move.jerk_factor;
			d^.axis_v_stop.Execute := TRUE;
			StateNext(d^.state);
		ELSE
			d^.state := State.RST_DONE;
		END_IF
	6:
		IF d^.axis_v_stop.Done THEN
			d^.axis_v_stop.Execute := FALSE;
			d^.axis_v_mabs.Execute := FALSE;
			d^.state := State.RST_DONE;
		END_IF
	//////\\
	////\\\\
	//\\\\\\
	State.HOME:
		d^.axis_spin.power^.bDriveStart := TRUE;
		d^.axis_spin.overload_check := TRUE;
		StateNext(d^.state);
	52:
		IF d^.axis_spin.power^.Status THEN
			d^.axis_spin_follow_data.target := d^.axis_move.ref;
			d^.axis_spin_follow_data.ratio := d^.μm_per_rev * 1E-3;
			d^.axis_spin_fb.follow(follow_data:= ADR(d^.axis_spin_follow_data), state:= 1);
			StateNext(d^.state);
		END_IF
	53:
		d^.axis_move.home_to_encoder := FALSE;
		d^.axis_move.state := State.HOME;
		StateNext(d^.state);
	54:
		IF d^.axis_move.state < 60 THEN // ignore set position phase
			d^.axis_spin_fb.follow(follow_data:= ADR(d^.axis_spin_follow_data), state:= 2);
		END_IF
		IF d^.axis_move.state = State.HOME_FORWARD THEN
			d^.axis_spin_fb.follow(follow_data:= ADR(d^.axis_spin_follow_data), state:= 1);
			StateNext(d^.state);
		END_IF
	55:
		d^.axis_spin_fb.follow(follow_data:= ADR(d^.axis_spin_follow_data), state:= 2);
		IF d^.axis_move.state = State.HOME_DONE THEN
			d^.axis_move.overload_check := TRUE;
			d^.state := State.HOME_DONE;
		END_IF
	//////\\
	////\\\\
	//\\\\\\
	State.HOME_OFFSET:
		d^.axis_move.home_offset_μ := 0;
		d^.axis_move.state := State.HOME_OFFSET;
		StateNext(d^.state);
	92:
		d^.axis_spin_fb.follow(follow_data:= ADR(d^.axis_spin_follow_data), state:= 2);
		IF d^.axis_move.state = State.HOME_OFFSET_DONE THEN
			d^.axis_move.state := State.READY;
			StateNext(d^.state);
		END_IF
	93:
		d^.axis_v_sp.Position := d^.axis_move.ref^.fAimPosition;
		d^.axis_v_sp.Execute := TRUE;
		StateNext(d^.state);
	94:
		IF d^.axis_v_sp.Done THEN
			d^.axis_v_sp.Execute := FALSE;
			StateNext(d^.state);
		END_IF
	95:
		d^.axis_move_follow_data.target := d^.axis_v;
		d^.axis_move_follow_data.ratio := 1.0;
		d^.axis_move_fb.follow(follow_data:= ADR(d^.axis_move_follow_data), state:= 1);
		d^.axis_spin_follow_data.target := d^.axis_v;
		d^.axis_spin_follow_data.ratio := d^.μm_per_rev * 1E-3;
		d^.axis_spin_fb.follow(follow_data:= ADR(d^.axis_spin_follow_data), state:= 1);
		d^.state := State.HOME_OFFSET_DONE;
	//////\\
	////\\\\
	//\\\\\\
	State.READY:
		d^.axis_move_fb.follow(follow_data:= ADR(d^.axis_move_follow_data), state:= 2);
		d^.axis_spin_fb.follow(follow_data:= ADR(d^.axis_spin_follow_data), state:= 2);
	//////\\
	////\\\\
	//\\\\\\
	State.RUN:
		IF d^.axis_move.state = State.READY THEN
			d^.axis_spin_fb.follow(follow_data:= ADR(d^.axis_spin_follow_data), state:= 1);
			d^.lubricate.on := TRUE;
			StateNext(d^.state);
		END_IF
	102:
		d^.axis_v_mabs.Position := d^.begin_μm;
		d^.axis_v_mabs.Velocity := d^.rps * d^.μm_per_rev;
		d^.axis_v_mabs.Acceleration := d^.axis_v_mabs.Velocity / d^.axis_move.ramp_time_sec;
		d^.axis_v_mabs.Deceleration := d^.axis_v_mabs.Acceleration;
		d^.axis_v_mabs.Jerk := d^.axis_v_mabs.Acceleration * d^.axis_move.jerk_factor;
		d^.axis_v_mabs.Execute := TRUE;
		StateNext(d^.state);
	103:
		d^.axis_move_fb.follow(follow_data:= ADR(d^.axis_move_follow_data), state:= 2);
		d^.axis_spin_fb.follow(follow_data:= ADR(d^.axis_spin_follow_data), state:= 2);
		IF d^.axis_v_mabs.Done THEN
			d^.axis_v_mabs.Execute := FALSE;
			StateNext(d^.state);
		END_IF
	104:
		d^.axis_v_mabs.Position := d^.begin_μm + d^.depth_μm;
		d^.axis_v_mabs.Velocity := d^.rps * d^.μm_per_rev;
		d^.axis_v_mabs.Acceleration := d^.axis_v_mabs.Velocity / d^.axis_move.ramp_time_sec;
		d^.axis_v_mabs.Deceleration := d^.axis_v_mabs.Acceleration;
		d^.axis_v_mabs.Jerk := d^.axis_v_mabs.Acceleration * d^.axis_move.jerk_factor;
		d^.axis_v_mabs.Execute := TRUE;
		StateNext(d^.state);
		d^.load_sum := 0;
		d^.load_count := 0;
	105:
		d^.axis_move_fb.follow(follow_data:= ADR(d^.axis_move_follow_data), state:= 2);
		d^.axis_spin_fb.follow(follow_data:= ADR(d^.axis_spin_follow_data), state:= 2);
		IF d^.axis_v_mabs.Done THEN
			d^.axis_v_mabs.Execute := FALSE;
			StateNext(d^.state);
		END_IF
		d^.load_sum := d^.load_sum + d^.axis_spin.torque_Nm_abs;
		d^.load_count := d^.load_count + 1;
		d^.load := (d^.load_sum / d^.load_count) / d^.axis_spin.torque_rated_Nm;
	106: // backlash compensate start
		d^.axis_spin_follow_data.offset_motion(
			state:= 1,
			tp:= d^.backlash_μ,
			tv:= d^.rps * 1E3,
			ta:= d^.rps * 1E3 / d^.axis_spin.ramp_time_sec,
			jerk_factor:= d^.axis_spin.jerk_factor);
		StateNext(d^.state);
	107: // backlash compensate
		d^.axis_spin_fb.follow(follow_data:= ADR(d^.axis_spin_follow_data), state:= 2);
		d^.axis_spin_follow_data.offset_motion(state:= 2, dt_sec:= d^.time_delta_sec);
		d^.axis_spin_follow_data.offset := d^.axis_spin_follow_data.offset_motion.p;
		IF ABS(d^.axis_spin_follow_data.offset) >= d^.backlash_μ THEN
			StateNext(d^.state);
		END_IF
	108:
		d^.axis_v_mabs.Position := d^.begin_μm;
		d^.axis_v_mabs.Velocity := d^.rps * d^.μm_per_rev;
		d^.axis_v_mabs.Acceleration := d^.axis_v_mabs.Velocity / d^.axis_move.ramp_time_sec;
		d^.axis_v_mabs.Deceleration := d^.axis_v_mabs.Acceleration;
		d^.axis_v_mabs.Jerk := d^.axis_v_mabs.Acceleration * d^.axis_move.jerk_factor;
		d^.axis_v_mabs.Execute := TRUE;
		StateNext(d^.state);
	109:
		d^.axis_move_fb.follow(follow_data:= ADR(d^.axis_move_follow_data), state:= 2);
		d^.axis_spin_fb.follow(follow_data:= ADR(d^.axis_spin_follow_data), state:= 2);
		IF d^.axis_v_mabs.Done THEN
			d^.axis_v_mabs.Execute := FALSE;
			StateNext(d^.state);
		END_IF
	110:
		d^.state := State.READY;
END_CASE

END_FUNCTION_BLOCK

// Device/Application/AxisFB
FUNCTION_BLOCK PUBLIC AxisFB
VAR_INPUT
	d: POINTER TO AxisEC;
END_VAR

d^.torque_Nm := d^.ref^.fActTorque;
d^.torque_Nm_abs := ABS(d^.torque_Nm);
// giá trị .fActTorque có thể khác nhau tuỳ PLC, trong trường hợp PLC Inovance này fActTorque là giá trị từ phần trăm moment
// 0.0% đến hơn 100.0%, nên phải nhân với .torque_rated_Nm đọc được ở hàm MAIN
d^.home_hit_timer(IN:= , PT:= , Q=> , ET=> );
// timer để lấy gốc, khi lùi về chạm gốc, giá trị moment sẽ tăng lên đến giá trị quy định (trong chương trình này là 1.27Nm)
// để tránh bị nhiễu thì moment quy định cần phải duy trì trong một thời gian mới có thể xác định gốc
d^.overload_hold_torque_timer(IN:= , PT:= , Q=> , ET=> );
// timer quá tải
IF d^.overload_check THEN
	d^.overload_hold_torque_timer.IN := d^.torque_Nm_abs > d^.overload_hold_torque_Nm;
	d^.overload := d^.overload_hold_torque_timer.Q OR d^.torque_Nm_abs > d^.overload_instant_torque_Nm;
END_IF
//////\\
////\\\\
//\\\\\\
d^.set_torque_limit(
	scale_factor:= d^.ref^.fScalefactor, 
	write:= d^.write, 
	torque_rated_Nm:= d^.torque_rated_Nm, 
	negative_Nm:= , 
	positive_Nm:= , 
	execute:= , 
	done=> );
CASE d^.state OF
	State.RST: // reset trục
		d^.read_status^.Enable := TRUE; // bật đọc trạng thái servo
		StateNext(d^.state);
	2:
		IF d^.read_status^.Valid THEN
			StateNext(d^.state);
		END_IF
	3:
		d^.inch^.InchBackward := FALSE;
		d^.inch^.InchForward := FALSE;
		d^.fsv^.bExecute := FALSE;
		d^.fsv^.fSetPosition := d^.ref^.fActPosition;
		d^.set_torque_limit.execute := FALSE;
		StateNext(d^.state);
	4:
		IF NOT d^.inch^.Busy AND NOT d^.fsv^.bError THEN
			StateNext(d^.state);
		END_IF
	5:
		IF d^.mabs^.Busy THEN // nếu hàm dịch chuyển MC_MoveAbsolute đang hoạt dộng thì kích hoạt hàm MC_Stop
			d^.stop^.Deceleration := d^.mabs^.Velocity / 0.01;
			d^.stop^.Jerk := d^.stop^.Deceleration * d^.jerk_factor;
			d^.stop^.Execute := TRUE;
			StateNext(d^.state);
		ELSE // nếu không thì nhảy đến bước tiếp theo
			d^.state := 21;
		END_IF
	6: // hàm SMC_Inch đang không hoạt động và hàm MC_Stop hoàn thành
		IF d^.stop^.Done THEN
			d^.state := 21;
		END_IF
	//
	21:
		d^.mabs^.Execute := FALSE; // sau khi các hàm hoàn thành, phải đặt biến Execute về FALSE
		d^.stop^.Execute := FALSE; // vì muốn chạy hàm cần có tín hiệu rising edge
		d^.power^.bDriveStart := FALSE; // tắt servo
		StateNext(d^.state);
	22:
		IF NOT d^.power^.Status THEN // đã tắt xong servo
			StateNext(d^.state);
		END_IF
	23:
		IF d^.read_status^.FBErrorOccured THEN // nếu có lỗi xảy ra thì xoá lỗi cũ
			SMC_ClearFBError(pDrive:= d^.ref); // xoá lỗi
			StateNext(d^.state);
		ELSE // nếu không có thì nhảy đến bước cuối
			d^.state := 31;
		END_IF
	24:
		IF d^.read_status^.FBErrorOccured THEN
			d^.reset^.Execute := TRUE; // reset lỗi
			StateNext(d^.state);
		END_IF
	25:
		IF d^.reset^.Done THEN
			d^.reset^.Execute := FALSE;
			SMC_ClearFBError(pDrive:= d^.ref); // xoá lỗi
			d^.state := 31;
		END_IF
	//
	31:
		d^.read_status^.Enable := FALSE;
		d^.state := State.RST_DONE;
	//////\\
	////\\\\
	//\\\\\\
	State.HOME:
		d^.power^.bDriveStart := TRUE; // bật servo để bắt đầu lấy gốc
		StateNext(d^.state);
	52:
		IF d^.power^.Status THEN // servo đã sẵn sàng
			StateNext(d^.state);
		END_IF
	53:
		IF d^.home_done THEN // đã lấy gốc trước đó thì nhảy đến bước HOME_FORWARD
			d^.state := State.HOME_FORWARD;
		ELSE // chưa lấy gốc thì qua bước tiếp theo
			IF d^.home_to_encoder THEN
				d^.state := 59;
			ELSE
				StateNext(d^.state);
			END_IF
		END_IF
	54:
		d^.set_mode^.nControllerMode := SMC_CONTROLLER_MODE.SMC_velocity;// chuyển chế độ servo sang tốc độ
		// ở chế độ .SMC_torque hoặc .SMC_velocity, khi servo vị chặn nó sẽ không vọt sau khi được nhả ra
		d^.set_mode^.bExecute := TRUE;
		StateNext(d^.state);
	55:
		IF d^.set_mode^.bDone THEN // chuyển chế độ xong
			d^.set_mode^.bExecute := FALSE;
			StateNext(d^.state);
		END_IF
	56:
		d^.set_torque_limit.negative_Nm := d^.home_torque_Nm;
		d^.set_torque_limit.positive_Nm := d^.home_torque_Nm;
		d^.set_torque_limit.execute := TRUE;
		StateNext(d^.state);
	57:
		IF d^.set_torque_limit.done THEN
			d^.set_torque_limit.execute := FALSE;
			StateNext(d^.state);
		END_IF
	58:
		d^.inch^.Velocity := d^.home_back_μ_per_sec; // lùi về
		d^.inch^.Distance := 1E16;
		d^.inch^.Acceleration := d^.inch^.Velocity / 0.1;
		d^.inch^.Deceleration := d^.inch^.Acceleration;
		d^.inch^.Jerk := d^.inch^.Acceleration * d^.jerk_factor;
		d^.inch^.InchBackward := TRUE; // .InchBackward là lùi
		d^.inch^.InchForward := FALSE; // .InchForward là tiến
		// nếu .InchBackward và .InchForward cùng bằng TRUE hoặc FALSE thì servo không chạy
		d^.home_hit_timer.IN := FALSE; // reset timer
		d^.home_hit_test := FALSE; // reset test
		StateNext(d^.state);
	59:
		d^.home_hit_timer.IN := d^.torque_Nm_abs >= d^.home_torque_Nm * 0.95 OR d^.home_hit_test; // set timer, * 0.95 để chắc ăn, tránh bị nhiễu
		IF d^.home_hit_timer.Q OR d^.home_to_encoder THEN // khi timer kích hoạt, dừng hàm SMC_Inch
			d^.inch^.InchBackward := FALSE;
			d^.inch^.InchForward := FALSE;
			d^.mabs^.Position := d^.ref^.fActPosition + d^.home_offset_absolute_μ;
			IF d^.home_encoder_value_recorded THEN
				calculate_home_delta_μ();
				d^.mabs^.Position := d^.mabs^.Position + d^.home_delta_μ;
			ELSE
				d^.home_encoder_value_save^ := d^.encoder_single_position;
				d^.home_encoder_value_recorded := TRUE;
			END_IF
			// gán tạm giá trị vào hàm MC_MoveAbsolute để đến bước tiếp theo
			// .fActPosition là vị trí thực tế của servo
			// ví dụ .fActPosition khi chạm là -123_000, có thể dùng "_" để phân cách các con số cho dễ đọc
			// .home_offset_absolute_micron = 1_000
			// d^.mabs^.Position sẽ bằng -123_000 + 1_000 = -122_000
			StateNext(d^.state);
		END_IF
	60:
		d^.sp^.Position := d^.ref^.fActPosition - d^.mabs^.Position;
		// thực hiện hàm MC_SetPosition để đưa giá trị .fActPosition về 0
		// bây giờ giá trị d^.sp^.Position = -123_000 - (-122_000) = -1_000
		// bây giờ servo đang ở vị trí va chạm, để về gốc thì nó phải dịch chuyển 1_000 micron
		// vậy vị trí gốc cách vị trí va chạm đúng bằng .home_offset_absolute_micron
		d^.sp^.Execute := TRUE;
		StateNext(d^.state);
	61:
		IF d^.sp^.Done THEN
			d^.sp^.Execute := FALSE;
			IF d^.max_μ_recorded THEN // đã có chiều dài trục -> tiến tới HOME_FORWARD
				d^.state := State.HOME_FORWARD;
			ELSE
				StateNext(d^.state); // tìm chiều dài trục
			END_IF
		END_IF
	62:
		d^.inch^.Velocity := d^.home_back_μ_per_sec; // tiến tới
		d^.inch^.Distance := 1E16;
		d^.inch^.Acceleration := d^.inch^.Velocity / 0.1;
		d^.inch^.Deceleration := d^.inch^.Acceleration;
		d^.inch^.Jerk := d^.inch^.Acceleration * d^.jerk_factor;
		d^.inch^.InchBackward := FALSE; // .InchBackward là lùi
		d^.inch^.InchForward := TRUE; // .InchForward là tiến
		// nếu .InchBackward và .InchForward cùng bằng TRUE hoặc FALSE thì servo không chạy
		d^.home_hit_timer.IN := FALSE; // reset timer
		d^.home_hit_test := FALSE; // reset test
		StateNext(d^.state);
	63:
		d^.home_hit_timer.IN := d^.torque_Nm_abs >= d^.home_torque_Nm * 0.95 OR d^.home_hit_test; // set timer, * 0.95 để chắc ăn, tránh bị nhiễu
		IF d^.home_hit_timer.Q THEN // khi timer kích hoạt, dừng hàm SMC_Inch
			d^.inch^.InchBackward := FALSE;
			d^.inch^.InchForward := FALSE;
			d^.max_μ := d^.ref^.fActPosition - d^.home_offset_absolute_μ;
			d^.max_μ_save^ := LREAL_TO_DINT(d^.max_μ);
			d^.max_μ_recorded := TRUE;
			d^.state := State.HOME_FORWARD;
		END_IF
	//////\\
	////\\\\
	//\\\\\\
	State.HOME_FORWARD:
		IF NOT d^.inch^.Busy THEN
			d^.set_mode^.nControllerMode := SMC_CONTROLLER_MODE.SMC_position; // set mode về điều khiển vị trí
			d^.set_mode^.bExecute := TRUE;
			StateNext(d^.state);
		END_IF
	72:
		IF d^.set_mode^.bDone THEN
			d^.set_mode^.bExecute := FALSE;
			StateNext(d^.state);
		END_IF
	73:
		// đưa giới hạn moment về 300%
		d^.set_torque_limit.negative_Nm := d^.torque_rated_Nm * 3.0;
		d^.set_torque_limit.positive_Nm := d^.torque_rated_Nm * 3.0;
		d^.set_torque_limit.execute := TRUE;
		StateNext(d^.state);
	74:
		IF d^.set_torque_limit.done THEN
			d^.set_torque_limit.execute := FALSE;
			StateNext(d^.state);
		END_IF
	75:
		// dịch chuyển tới vị trí gốc
		IF d^.home_done AND d^.home_done_forward_ignore THEN
			d^.mabs^.Position := d^.ref^.fActPosition;
		ELSE
			d^.mabs^.Position := 0;
		END_IF
		d^.mabs^.Velocity := d^.home_forward_μ_per_sec;
		d^.mabs^.Acceleration := d^.mabs^.Velocity / d^.ramp_time_sec;
		d^.mabs^.Deceleration := d^.mabs^.Acceleration;
		d^.mabs^.Jerk := d^.mabs^.Acceleration * d^.jerk_factor;
		d^.mabs^.Direction := MC_DIRECTION.shortest; // nếu là trục module, di chuyển đến vị trí gần nhất
		d^.mabs^.Execute := TRUE;
		StateNext(d^.state);
	76:
		IF d^.mabs^.Done THEN
			d^.mabs^.Execute := FALSE;
			d^.home_done := TRUE;
			d^.state := State.HOME_DONE;
		END_IF
	//////\\
	////\\\\
	//\\\\\\
	State.HOME_OFFSET: // địch chuyển tới vị trí HOME_OFFSET
		d^.mabs^.Position := d^.home_offset_μ;
		d^.mabs^.Velocity := d^.home_forward_μ_per_sec;
		d^.mabs^.Acceleration := d^.mabs^.Velocity / d^.ramp_time_sec;
		d^.mabs^.Deceleration := d^.mabs^.Acceleration;
		d^.mabs^.Jerk := d^.mabs^.Acceleration * d^.jerk_factor; // jerk chỉ có tác dụng khi Velocity ramp type khác Trapezoid
		d^.mabs^.Execute := TRUE;
		StateNext(d^.state);
	92:
		IF d^.mabs^.Done THEN // dịch chuyển xong
			d^.mabs^.Execute := FALSE;
			StateNext(d^.state);
		END_IF
	93:
		CASE d^.jog_type OF
			JogType.FSV:
				d^.jog_delta := 0;
				d^.fsv^.dwValueMask := UDINT_TO_DWORD(1 + 2 + 4 + 8);
				d^.fsv^.fSetPosition := d^.home_offset_μ;
				d^.fsv^.fSetVelocity := 0;
				d^.fsv^.fSetAcceleration := 0;
				d^.fsv^.fSetJerk := 0;
				d^.fsv^.bExecute := TRUE;
		END_CASE
		d^.state := State.HOME_OFFSET_DONE;
	//////\\
	////\\\\
	//\\\\\\
	State.READY:
		CASE d^.jog_type OF
			JogType.INCH:
				d^.inch^.Velocity := MIN(d^.max_μ_per_sec, d^.jog_velocity);
				d^.inch^.Acceleration := d^.jog_velocity / d^.ramp_time_sec;
				d^.inch^.Deceleration := d^.inch^.Acceleration;
				d^.inch^.Jerk := d^.inch^.Acceleration * d^.jerk_factor;
				d^.inch^.InchBackward := d^.jog_delta < 0;
				d^.inch^.InchForward := d^.jog_delta > 0;
				IF d^.inch^.InchBackward THEN
					d^.inch^.Distance := d^.ref^.fActPosition;
				END_IF
				IF d^.inch^.InchForward THEN
					d^.inch^.Distance := d^.max_μ - d^.ref^.fActPosition;
				END_IF
			JogType.FSV:
				IF d^.fsv^.bExecute AND NOT d^.fsv^.bError THEN
					d^.fsv^.fSetPosition := MAX(0, MIN(d^.max_μ, d^.fsv^.fSetPosition + d^.jog_delta));
					d^.fsv^.fSetVelocity := MIN(d^.max_μ_per_sec, ABS(d^.jog_velocity));
					d^.fsv^.fSetAcceleration := MIN(d^.max_μ_per_sec * 10, ABS(d^.jog_acceleration));
					d^.fsv^.fSetJerk := d^.fsv^.fSetAcceleration * d^.jerk_factor;
				END_IF
				d^.jog_delta := 0;
		END_CASE
	//////\\
	////\\\\
	//\\\\\\
	State.RUN:
		IF d^.fsv^.bExecute THEN
			d^.fsv^.bExecute := FALSE;
			StateNext(d^.state);
		ELSE
			d^.state := 103;
		END_IF
	102:
		IF NOT d^.fsv^.bError THEN
			StateNext(d^.state);
		END_IF
	103:
		// lệnh chạy đến vị trí chỉ định
		// xem hàm cut() và supply()
		// set d^.target_position_micron và d^.target_velocity_micron_per_sec sau đó set d^.state = State.RUN
		d^.mabs^.Position := MAX(0, MIN(d^.max_μ, d^.target_position_μ)); // giới hạn vị trí, xem save_apply()
		d^.mabs^.Velocity := MAX(0_100, MIN(d^.max_μ_per_sec, d^.target_velocity_μ_per_sec)); // giới hạn tốc độ, xem save_apply()
		d^.mabs^.Acceleration := d^.mabs^.Velocity / d^.ramp_time_sec;
		d^.mabs^.Deceleration := d^.mabs^.Acceleration;
		d^.mabs^.Jerk := d^.mabs^.Acceleration * d^.jerk_factor;
		d^.mabs^.Execute := TRUE;
		StateNext(d^.state);
	104:
		IF d^.mabs^.Done THEN
			d^.mabs^.Execute := FALSE;
			d^.state := State.READY;
		END_IF
END_CASE

ACTION calculate_home_delta_μ:
d^.home_encoder_delta := d^.home_encoder_value_save^ - d^.encoder_single_position;
IF d^.home_encoder_delta >= 0 THEN
	d^.home_delta_μ := ABS(d^.home_encoder_delta) / d^.ref^.fScalefactor;
ELSIF ABS(d^.home_encoder_delta) > (d^.encoder_resolution / 2) THEN
	d^.home_delta_μ := (d^.encoder_resolution - ABS(d^.home_encoder_delta)) / d^.ref^.fScalefactor;
ELSE
	d^.home_delta_μ := -ABS(d^.home_encoder_delta) / d^.ref^.fScalefactor;
END_IF
END_ACTION

METHOD follow
VAR_INPUT
	state: INT;
	follow_data: POINTER TO AxisECFollow;
END_VAR
CASE state OF
	1: // start follow
		follow_data^.self_begin := d^.ref^.fActPosition;
		follow_data^.target_begin := follow_data^.target^.fActPosition;
		follow_data^.offset := 0;
		follow_data^.deviation := 0;
		d^.fsv^.dwValueMask := UDINT_TO_DWORD(1 + 2 + 4 + 8);
		d^.fsv^.fSetPosition := follow_data^.self_begin;
		d^.fsv^.fSetVelocity := 0;
		d^.fsv^.fSetAcceleration := 0;
		d^.fsv^.fSetJerk := 0;
		d^.fsv^.bExecute := TRUE;
	2: // follow
		follow_data^.target_delta := follow_data^.target^.fActPosition - follow_data^.target_begin;
		d^.fsv^.fSetPosition := (follow_data^.self_begin - follow_data^.offset) + (follow_data^.target_delta / follow_data^.ratio);
		d^.fsv^.fSetVelocity := follow_data^.target^.fActVelocity / follow_data^.ratio;
		d^.fsv^.fSetAcceleration := follow_data^.target^.fActAcceleration / follow_data^.ratio;
		d^.fsv^.fSetJerk := follow_data^.target^.fActJerk / follow_data^.ratio;
		follow_data^.deviation := follow_data^.target_delta - (d^.ref^.fActPosition - follow_data^.self_begin + follow_data^.offset) * follow_data^.ratio;
END_CASE
END_METHOD

END_FUNCTION_BLOCK

// Device/Application/SimpleMotion
FUNCTION_BLOCK SimpleMotion
VAR_INPUT
	state: INT;
	tp: LREAL;
	tv: LREAL;
	ta: LREAL;
	jerk_factor: LREAL;
	dt_sec: LREAL;
END_VAR
VAR_OUTPUT
	p: LREAL;
	v: LREAL;
	a: LREAL;
	d: LREAL;
END_VAR

CASE state OF
	1:
		a := 0;
		v := 0;
		p := 0;
		d := 1;
	2:
		a := MIN(a + d * ta * jerk_factor * dt_sec, ta);
		v := MIN(v + d * a * dt_sec, tv);
		p := MIN(p + v * dt_sec, tp);
		IF p > 0.55 * tp THEN
			d := -1;
		END_IF
END_CASE

END_FUNCTION_BLOCK

// Device/Application/AxisFBSetTorqueLimit
FUNCTION_BLOCK AxisFBSetTorqueLimit
VAR_INPUT
	scale_factor: LREAL;
	write: POINTER TO SMC3_ETC_WriteParameter_CoE;
	torque_rated_Nm: LREAL;
	negative_Nm: LREAL;
	positive_Nm: LREAL;
	execute: BOOL;
END_VAR
VAR_OUTPUT
	execute_rise: R_TRIG;
	state: INT;
	done: BOOL;
END_VAR

execute_rise(CLK:= execute, Q=> );
IF execute_rise.Q THEN
	state := 1;
END_IF
IF execute THEN
	CASE state OF
		1:
			done := FALSE;
			IF scale_factor > 0 THEN
				write^.uiIndex := 16#60E1; // servo negative torque limit
			ELSE
				write^.uiIndex := 16#60E0; // servo positive torque limit
			END_IF
			write^.usiSubIndex := 0;
			write^.usiDataLength := 2;
			write^.dwValue := LREAL_TO_DWORD(1000 * (negative_Nm / torque_rated_Nm));
			write^.xExecute := TRUE;
			StateNext(state);
		2:
			IF write^.xDone THEN
				write^.xExecute := FALSE;
				StateNext(state);
			END_IF
		3:
			IF scale_factor > 0 THEN
				write^.uiIndex := 16#60E0; // servo positive torque limit
			ELSE
				write^.uiIndex := 16#60E1; // servo negative torque limit
			END_IF
			write^.usiSubIndex := 0;
			write^.usiDataLength := 2;
			write^.dwValue := LREAL_TO_DWORD(1000 * (positive_Nm / torque_rated_Nm));
			write^.xExecute := TRUE;
			StateNext(state);
		4:
			IF write^.xDone THEN
				write^.xExecute := FALSE;
				done := TRUE;
				state := 0;
			END_IF
	END_CASE
END_IF

END_FUNCTION_BLOCK

// Device/Application/Visualization
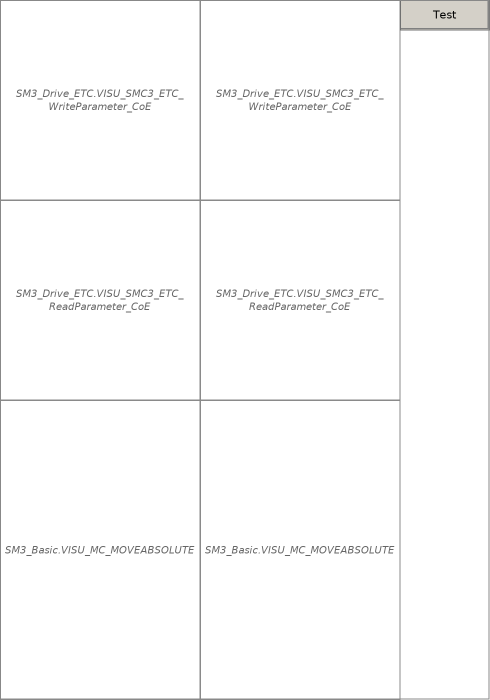
VISUALIZATION Visualization  // 490x700
    Frame (0,0 200x200)
        shows SM3_Drive_ETC.VISU_SMC3_ETC_WriteParameter_CoE(m_Input_FB := M.axiss_write[0])
    Frame (0,200 200x200)
        shows SM3_Drive_ETC.VISU_SMC3_ETC_ReadParameter_CoE(m_Input_FB := M.axiss_read[0])
    Frame (200,200 200x200)
        shows SM3_Drive_ETC.VISU_SMC3_ETC_ReadParameter_CoE(m_Input_FB := M.axiss_read[1])
    Frame (200,0 200x200)
        shows SM3_Drive_ETC.VISU_SMC3_ETC_WriteParameter_CoE(m_Input_FB := M.axiss_write[1])
    Button (400,0 90x30), "Test"
        toggle M.test
    Frame (0,400 200x300)
        shows SM3_Basic.VISU_MC_MOVEABSOLUTE(m_Input_FB := M.axiss_mabs[0])
    Frame (200,400 200x300)
        shows SM3_Basic.VISU_MC_MOVEABSOLUTE(m_Input_FB := M.axiss_mabs[1])
END_VISUALIZATION
